LIN {X -0.031,Y -424.133,Z 625.479,A 0.000,B 0.000,C 90.000,E1 266.216} C_DIS
LIN {X -0.178,Y -415.760,Z 625.479,A 0.000,B 0.000,C 90.000,E1 266.159} C_DIS
LIN {X 0.095,Y -410.358,Z 625.478,A 0.000,B 0.000,C 90.000,E1 266.102} C_DIS
LIN {X 0.011,Y -180.925,Z 625.478,A 0.000,B 0.000,C 90.000,E1 266.102} C_DIS
LIN {X -0.004,Y -180.875,Z 625.473,A 0.000,B 0.000,C 90.000,E1 265.065} C_DIS
LIN {X 0.078,Y -178.941,Z 625.443,A 0.000,B 0.000,C 90.000,E1 259.803} C_DIS
LIN {X -0.054,Y -175.991,Z 625.415,A 0.000,B 0.000,C 90.000,E1 254.755} C_DIS
LIN {X 0.061,Y -175.493,Z 625.410,A 0.000,B 0.000,C 90.000,E1 253.866} C_DIS
LIN {X -0.045,Y -172.236,Z 625.387,A 0.000,B 0.000,C 90.000,E1 249.625} C_DIS
LIN {X -0.066,Y -171.714,Z 625.382,A 0.000,B 0.000,C 90.000,E1 248.773} C_DIS
LIN {X 0.019,Y -167.309,Z 625.353,A 0.000,B 0.000,C 90.000,E1 243.563} C_DIS
LIN {X 0.024,Y -166.690,Z 625.348,A 0.000,B 0.000,C 90.000,E1 242.692} C_DIS
LIN {X 0.015,Y -162.671,Z 625.324,A 0.000,B 0.000,C 90.000,E1 238.329} C_DIS
LIN {X -0.012,Y -161.361,Z 625.314,A 0.000,B 0.000,C 90.000,E1 236.580} C_DIS
LIN {X 0.022,Y -157.354,Z 625.290,A 0.000,B 0.000,C 90.000,E1 232.145} C_DIS
LIN {X 0.051,Y -155.342,Z 625.275,A 0.000,B 0.000,C 90.000,E1 229.461} C_DIS
LIN {X -0.020,Y -151.690,Z 625.250,A 0.000,B 0.000,C 90.000,E1 225.000} C_DIS
LIN {X 0.028,Y -150.553,Z 625.240,A 0.000,B 0.000,C 90.000,E1 223.176} C_DIS
LIN {X -0.054,Y -147.279,Z 625.215,A 0.000,B 0.000,C 90.000,E1 218.669} C_DIS
LIN {X 0.033,Y -145.307,Z 625.194,A 0.000,B 0.000,C 90.000,E1 214.978} C_DIS
LIN {X 0.025,Y -142.398,Z 625.164,A 0.000,B 0.000,C 90.000,E1 209.461} C_DIS
LIN {X 0.008,Y -141.380,Z 625.148,A 0.000,B 0.000,C 90.000,E1 206.693} C_DIS
LIN {X 0.049,Y -139.349,Z 625.112,A 0.000,B 0.000,C 90.000,E1 200.174} C_DIS
LIN {X -0.009,Y -138.785,Z 625.097,A 0.000,B 0.000,C 90.000,E1 197.402} C_DIS
LIN {X 0.049,Y -138.344,Z 625.055,A 0.000,B 0.000,C 90.000,E1 189.905} C_DIS
LIN {X 0.069,Y -139.387,Z 625.008,A 0.000,B 0.000,C 90.000,E1 181.489} C_DIS
LIN {X -0.017,Y -141.284,Z 624.972,A 0.000,B 0.000,C 90.000,E1 175.008} C_DIS
LIN {X -0.059,Y -142.647,Z 624.957,A 0.000,B 0.000,C 90.000,E1 172.243} C_DIS
LIN {X 0.033,Y -144.984,Z 624.931,A 0.000,B 0.000,C 90.000,E1 167.589} C_DIS
LIN {X 0.023,Y -147.611,Z 624.911,A 0.000,B 0.000,C 90.000,E1 163.921} C_DIS
LIN {X -0.040,Y -150.234,Z 624.890,A 0.000,B 0.000,C 90.000,E1 160.296} C_DIS
LIN {X -0.025,Y -153.627,Z 624.870,A 0.000,B 0.000,C 90.000,E1 156.666} C_DIS
LIN {X -0.037,Y -157.042,Z 624.850,A 0.000,B 0.000,C 90.000,E1 153.076} C_DIS
LIN {X 0.033,Y -161.168,Z 624.831,A 0.000,B 0.000,C 90.000,E1 149.488} C_DIS
LIN {X -0.024,Y -163.264,Z 624.821,A 0.000,B 0.000,C 90.000,E1 147.740} C_DIS
LIN {X 0.074,Y -167.704,Z 624.801,A 0.000,B 0.000,C 90.000,E1 144.196} C_DIS
LIN {X -0.012,Y -171.524,Z 624.787,A 0.000,B 0.000,C 90.000,E1 141.618} C_DIS
LIN {X 0.030,Y -176.462,Z 624.768,A 0.000,B 0.000,C 90.000,E1 138.162} C_DIS
LIN {X -0.099,Y -180.758,Z 624.753,A 0.000,B 0.000,C 90.000,E1 135.648} C_DIS
LIN {X 0.019,Y -186.164,Z 624.735,A 0.000,B 0.000,C 90.000,E1 132.243} C_DIS
LIN {X -0.012,Y -191.121,Z 624.720,A 0.000,B 0.000,C 90.000,E1 129.564} C_DIS
LIN {X -0.069,Y -287.980,Z 624.720,A 0.000,B 0.000,C 90.000,E1 129.564} C_DIS
LIN {X -0.120,Y -289.136,Z 624.720,A 0.000,B 0.000,C 90.000,E1 129.564} C_DIS
LIN {X -0.085,Y -293.449,Z 624.719,A 0.000,B 0.000,C 90.000,E1 129.402} C_DIS
LIN {X 0.178,Y -295.651,Z 624.718,A 0.000,B 0.000,C 90.000,E1 129.197} C_DIS
LIN {X 0.065,Y -298.660,Z 624.716,A 0.000,B 0.000,C 90.000,E1 128.910} C_DIS
LIN {X 0.032,Y -302.298,Z 624.713,A 0.000,B 0.000,C 90.000,E1 128.338} C_DIS
LIN {X -0.020,Y -303.752,Z 624.711,A 0.000,B 0.000,C 90.000,E1 128.016} C_DIS
LIN {X -0.020,Y -304.897,Z 624.709,A 0.000,B 0.000,C 90.000,E1 127.684} C_DIS
LIN {X 0.096,Y -315.476,Z 624.689,A 0.000,B 0.000,C 90.000,E1 124.072} C_DIS
LIN {X -0.022,Y -325.465,Z 624.673,A 0.000,B 0.000,C 90.000,E1 121.209} C_DIS
LIN {X 0.087,Y -336.777,Z 624.658,A 0.000,B 0.000,C 90.000,E1 118.359} C_DIS
LIN {X 0.035,Y -349.518,Z 624.642,A 0.000,B 0.000,C 90.000,E1 115.591} C_DIS
LIN {X -0.166,Y -362.130,Z 624.629,A 0.000,B 0.000,C 90.000,E1 113.206} C_DIS
LIN {X 0.145,Y -376.051,Z 624.616,A 0.000,B 0.000,C 90.000,E1 110.791} C_DIS
LIN {X 0.066,Y -391.379,Z 624.603,A 0.000,B 0.000,C 90.000,E1 108.489} C_DIS
LIN {X -0.135,Y -408.226,Z 624.590,A 0.000,B 0.000,C 90.000,E1 106.260} C_DIS
LIN {X -0.165,Y -426.717,Z 624.578,A 0.000,B 0.000,C 90.000,E1 104.064} C_DIS
LIN {X -0.079,Y -446.611,Z 624.566,A 0.000,B 0.000,C 90.000,E1 101.951} C_DIS
LIN {X -0.051,Y -467.104,Z 624.556,A 0.000,B 0.000,C 90.000,E1 100.018} C_DIS
LIN {X -0.014,Y -472.187,Z 624.553,A 0.000,B 0.000,C 90.000,E1 99.557} C_DIS
LIN {X 0.000,Y -474.149,Z 624.552,A 0.000,B 0.000,C 90.000,E1 99.321} C_DIS
LIN {X -0.064,Y -475.647,Z 624.550,A 0.000,B 0.000,C 90.000,E1 99.095} C_DIS
LIN {X -0.200,Y -476.871,Z 624.549,A 0.000,B 0.000,C 90.000,E1 98.859} C_DIS
LIN {X 0.135,Y -477.767,Z 624.548,A 0.000,B 0.000,C 90.000,E1 98.568} C_DIS
LIN {X -0.197,Y -478.729,Z 624.545,A 0.000,B 0.000,C 90.000,E1 98.106} C_DIS
LIN {X -0.049,Y -478.707,Z 624.542,A 0.000,B 0.000,C 90.000,E1 97.587} C_DIS
LIN {X 0.106,Y -477.700,Z 624.539,A 0.000,B 0.000,C 90.000,E1 97.068} C_DIS
LIN {X -0.024,Y -476.783,Z 624.538,A 0.000,B 0.000,C 90.000,E1 96.834} C_DIS
LIN {X -0.212,Y -475.534,Z 624.537,A 0.000,B 0.000,C 90.000,E1 96.606} C_DIS
LIN {X -0.214,Y -470.227,Z 624.532,A 0.000,B 0.000,C 90.000,E1 95.853} C_DIS
LIN {X 0.070,Y -456.360,Z 624.521,A 0.000,B 0.000,C 90.000,E1 93.784} C_DIS
LIN {X 0.196,Y -442.672,Z 624.508,A 0.000,B 0.000,C 90.000,E1 91.432} C_DIS
LIN {X 0.081,Y -432.630,Z 624.498,A 0.000,B 0.000,C 90.000,E1 89.599} C_DIS
LIN {X -0.058,Y -425.082,Z 624.490,A 0.000,B 0.000,C 90.000,E1 88.282} C_DIS
LIN {X -0.169,Y -415.676,Z 624.481,A 0.000,B 0.000,C 90.000,E1 86.674} C_DIS
LIN {X -0.133,Y -400.162,Z 624.466,A 0.000,B 0.000,C 90.000,E1 83.913} C_DIS
LIN {X -0.126,Y -386.762,Z 624.452,A 0.000,B 0.000,C 90.000,E1 81.376} C_DIS
LIN {X 0.075,Y -372.503,Z 624.436,A 0.000,B 0.000,C 90.000,E1 78.465} C_DIS
LIN {X 0.060,Y -361.513,Z 624.423,A 0.000,B 0.000,C 90.000,E1 76.117} C_DIS
LIN {X -0.050,Y -347.259,Z 624.405,A 0.000,B 0.000,C 90.000,E1 72.834} C_DIS
LIN {X 0.039,Y -336.337,Z 624.389,A 0.000,B 0.000,C 90.000,E1 70.061} C_DIS
LIN {X 0.095,Y -324.067,Z 624.370,A 0.000,B 0.000,C 90.000,E1 66.613} C_DIS
LIN {X -0.068,Y -314.012,Z 624.352,A 0.000,B 0.000,C 90.000,E1 63.461} C_DIS
LIN {X 0.025,Y -304.661,Z 624.334,A 0.000,B 0.000,C 90.000,E1 60.205} C_DIS
LIN {X 0.025,Y -295.894,Z 624.316,A 0.000,B 0.000,C 90.000,E1 56.914} C_DIS
LIN {X -0.010,Y -287.671,Z 624.298,A 0.000,B 0.000,C 90.000,E1 53.577} C_DIS
LIN {X -0.099,Y -281.225,Z 624.283,A 0.000,B 0.000,C 90.000,E1 50.884} C_DIS
LIN {X 0.000,Y -276.089,Z 624.271,A 0.000,B 0.000,C 90.000,E1 48.809} C_DIS
LIN {X 0.175,Y -272.365,Z 624.263,A 0.000,B 0.000,C 90.000,E1 47.391} C_DIS
LIN {X -0.075,Y -268.402,Z 624.256,A 0.000,B 0.000,C 90.000,E1 46.053} C_DIS
LIN {X -0.067,Y -261.947,Z 624.244,A 0.000,B 0.000,C 90.000,E1 43.947} C_DIS
LIN {X 0.019,Y -253.976,Z 624.230,A 0.000,B 0.000,C 90.000,E1 41.434} C_DIS
LIN {X -0.009,Y -244.166,Z 624.212,A 0.000,B 0.000,C 90.000,E1 38.177} C_DIS
LIN {X -0.027,Y -236.115,Z 624.196,A 0.000,B 0.000,C 90.000,E1 35.231} C_DIS
LIN {X 0.061,Y -228.843,Z 624.179,A 0.000,B 0.000,C 90.000,E1 32.212} C_DIS
LIN {X 0.032,Y -220.667,Z 624.158,A 0.000,B 0.000,C 90.000,E1 28.409} C_DIS
LIN {X -0.044,Y -214.977,Z 624.141,A 0.000,B 0.000,C 90.000,E1 25.335} C_DIS
LIN {X -0.012,Y -208.974,Z 624.119,A 0.000,B 0.000,C 90.000,E1 21.408} C_DIS
LIN {X -0.072,Y -204.153,Z 624.097,A 0.000,B 0.000,C 90.000,E1 17.457} C_DIS
LIN {X 0.061,Y -200.407,Z 624.075,A 0.000,B 0.000,C 90.000,E1 13.411} C_DIS
LIN {X 0.038,Y -197.242,Z 624.048,A 0.000,B 0.000,C 90.000,E1 8.568} C_DIS
LIN {X 0.032,Y -197.987,Z 623.952,A 0.000,B 0.000,C 90.000,E1 351.376} C_DIS
LIN {X 0.025,Y -201.441,Z 623.925,A 0.000,B 0.000,C 90.000,E1 346.520} C_DIS
LIN {X 0.072,Y -205.463,Z 623.903,A 0.000,B 0.000,C 90.000,E1 342.489} C_DIS
LIN {X -0.041,Y -210.309,Z 623.881,A 0.000,B 0.000,C 90.000,E1 338.539} C_DIS
LIN {X 0.002,Y -215.908,Z 623.859,A 0.000,B 0.000,C 90.000,E1 334.588} C_DIS
LIN {X -0.073,Y -222.153,Z 623.837,A 0.000,B 0.000,C 90.000,E1 330.717} C_DIS
LIN {X 0.101,Y -229.051,Z 623.816,A 0.000,B 0.000,C 90.000,E1 326.834} C_DIS
LIN {X -0.003,Y -235.031,Z 623.799,A 0.000,B 0.000,C 90.000,E1 323.829} C_DIS
LIN {X 0.095,Y -242.933,Z 623.778,A 0.000,B 0.000,C 90.000,E1 320.070} C_DIS
LIN {X -0.013,Y -251.590,Z 623.758,A 0.000,B 0.000,C 90.000,E1 316.419} C_DIS
LIN {X -0.035,Y -261.286,Z 623.738,A 0.000,B 0.000,C 90.000,E1 312.813} C_DIS
LIN {X 0.019,Y -270.004,Z 623.722,A 0.000,B 0.000,C 90.000,E1 309.967} C_DIS
LIN {X -0.030,Y -282.468,Z 623.703,A 0.000,B 0.000,C 90.000,E1 306.503} C_DIS
LIN {X 0.103,Y -296.445,Z 623.684,A 0.000,B 0.000,C 90.000,E1 303.086} C_DIS
LIN {X 0.049,Y -312.049,Z 623.666,A 0.000,B 0.000,C 90.000,E1 299.795} C_DIS
LIN {X -0.073,Y -327.245,Z 623.649,A 0.000,B 0.000,C 90.000,E1 296.924} C_DIS
LIN {X 0.087,Y -344.942,Z 623.632,A 0.000,B 0.000,C 90.000,E1 293.770} C_DIS
LIN {X -0.016,Y -360.212,Z 623.619,A 0.000,B 0.000,C 90.000,E1 291.354} C_DIS
LIN {X 0.111,Y -378.973,Z 623.604,A 0.000,B 0.000,C 90.000,E1 288.671} C_DIS
LIN {X 0.178,Y -399.589,Z 623.589,A 0.000,B 0.000,C 90.000,E1 286.079} C_DIS
LIN {X 0.017,Y -413.489,Z 623.580,A 0.000,B 0.000,C 90.000,E1 284.426} C_DIS
LIN {X -0.050,Y -424.647,Z 623.573,A 0.000,B 0.000,C 90.000,E1 283.063} C_DIS
LIN {X -0.045,Y -435.361,Z 623.565,A 0.000,B 0.000,C 90.000,E1 281.715} C_DIS
LIN {X 0.112,Y -445.670,Z 623.558,A 0.000,B 0.000,C 90.000,E1 280.366} C_DIS
LIN {X 0.083,Y -457.496,Z 623.549,A 0.000,B 0.000,C 90.000,E1 278.803} C_DIS
LIN {X -0.025,Y -466.986,Z 623.542,A 0.000,B 0.000,C 90.000,E1 277.530} C_DIS
LIN {X -0.112,Y -472.142,Z 623.538,A 0.000,B 0.000,C 90.000,E1 276.777} C_DIS
LIN {X -0.006,Y -475.183,Z 623.535,A 0.000,B 0.000,C 90.000,E1 276.258} C_DIS
LIN {X 0.120,Y -477.839,Z 623.532,A 0.000,B 0.000,C 90.000,E1 275.739} C_DIS
LIN {X -0.215,Y -480.121,Z 623.529,A 0.000,B 0.000,C 90.000,E1 275.277} C_DIS
LIN {X -0.062,Y -482.024,Z 623.526,A 0.000,B 0.000,C 90.000,E1 274.759} C_DIS
LIN {X 0.062,Y -483.545,Z 623.524,A 0.000,B 0.000,C 90.000,E1 274.245} C_DIS
LIN {X 0.234,Y -484.683,Z 623.521,A 0.000,B 0.000,C 90.000,E1 273.726} C_DIS
LIN {X -0.100,Y -485.485,Z 623.518,A 0.000,B 0.000,C 90.000,E1 273.269} C_DIS
LIN {X 0.084,Y -485.991,Z 623.515,A 0.000,B 0.000,C 90.000,E1 272.751} C_DIS
LIN {X -0.237,Y -486.190,Z 623.513,A 0.000,B 0.000,C 90.000,E1 272.293} C_DIS
LIN {X -0.051,Y -486.080,Z 623.510,A 0.000,B 0.000,C 90.000,E1 271.776} C_DIS
LIN {X 0.118,Y -485.598,Z 623.507,A 0.000,B 0.000,C 90.000,E1 271.260} C_DIS
LIN {X -0.196,Y -484.736,Z 623.504,A 0.000,B 0.000,C 90.000,E1 270.802} C_DIS
LIN {X -0.027,Y -483.413,Z 623.502,A 0.000,B 0.000,C 90.000,E1 270.286} C_DIS
LIN {X 0.136,Y -481.532,Z 623.499,A 0.000,B 0.000,C 90.000,E1 269.771} C_DIS
LIN {X -0.189,Y -478.902,Z 623.496,A 0.000,B 0.000,C 90.000,E1 269.312} C_DIS
LIN {X 0.118,Y -477.369,Z 623.495,A 0.000,B 0.000,C 90.000,E1 269.026} C_DIS
LIN {X -0.230,Y -473.473,Z 623.492,A 0.000,B 0.000,C 90.000,E1 268.568} C_DIS
LIN {X 0.064,Y -471.160,Z 623.490,A 0.000,B 0.000,C 90.000,E1 268.282} C_DIS
LIN {X -0.109,Y -468.523,Z 623.489,A 0.000,B 0.000,C 90.000,E1 268.051} C_DIS
LIN {X 0.217,Y -462.608,Z 623.486,A 0.000,B 0.000,C 90.000,E1 267.535} C_DIS
LIN {X -0.198,Y -459.195,Z 623.485,A 0.000,B 0.000,C 90.000,E1 267.364} C_DIS
LIN {X 0.042,Y -452.155,Z 623.483,A 0.000,B 0.000,C 90.000,E1 266.963} C_DIS
LIN {X 0.003,Y -444.697,Z 623.482,A 0.000,B 0.000,C 90.000,E1 266.674} C_DIS
LIN {X 0.010,Y -437.024,Z 623.480,A 0.000,B 0.000,C 90.000,E1 266.445} C_DIS
LIN {X 0.005,Y -428.475,Z 623.479,A 0.000,B 0.000,C 90.000,E1 266.274} C_DIS
LIN {X -0.014,Y -419.041,Z 623.479,A 0.000,B 0.000,C 90.000,E1 266.159} C_DIS
LIN {X 0.112,Y -411.810,Z 623.478,A 0.000,B 0.000,C 90.000,E1 266.102} C_DIS
LIN {X 0.018,Y -180.925,Z 623.478,A 0.000,B 0.000,C 90.000,E1 266.102} C_DIS
LIN {X -0.019,Y -180.899,Z 623.474,A 0.000,B 0.000,C 90.000,E1 265.241} C_DIS
LIN {X -0.069,Y -180.215,Z 623.464,A 0.000,B 0.000,C 90.000,E1 263.571} C_DIS
LIN {X 0.061,Y -179.034,Z 623.445,A 0.000,B 0.000,C 90.000,E1 260.151} C_DIS
LIN {X -0.052,Y -178.692,Z 623.441,A 0.000,B 0.000,C 90.000,E1 259.342} C_DIS
LIN {X 0.057,Y -175.741,Z 623.412,A 0.000,B 0.000,C 90.000,E1 254.212} C_DIS
LIN {X 0.053,Y -171.925,Z 623.384,A 0.000,B 0.000,C 90.000,E1 249.082} C_DIS
LIN {X 0.028,Y -171.298,Z 623.379,A 0.000,B 0.000,C 90.000,E1 248.230} C_DIS
LIN {X 0.073,Y -167.560,Z 623.355,A 0.000,B 0.000,C 90.000,E1 243.896} C_DIS
LIN {X 0.086,Y -166.186,Z 623.345,A 0.000,B 0.000,C 90.000,E1 242.153} C_DIS
LIN {X 0.076,Y -162.955,Z 623.326,A 0.000,B 0.000,C 90.000,E1 238.663} C_DIS
LIN {X -0.100,Y -160.863,Z 623.311,A 0.000,B 0.000,C 90.000,E1 236.087} C_DIS
LIN {X 0.100,Y -157.638,Z 623.292,A 0.000,B 0.000,C 90.000,E1 232.477} C_DIS
LIN {X 0.038,Y -155.676,Z 623.277,A 0.000,B 0.000,C 90.000,E1 229.828} C_DIS
LIN {X -0.017,Y -151.943,Z 623.252,A 0.000,B 0.000,C 90.000,E1 225.364} C_DIS
LIN {X -0.006,Y -150.181,Z 623.237,A 0.000,B 0.000,C 90.000,E1 222.651} C_DIS
LIN {X 0.023,Y -146.955,Z 623.212,A 0.000,B 0.000,C 90.000,E1 218.096} C_DIS
LIN {X 0.011,Y -145.542,Z 623.196,A 0.000,B 0.000,C 90.000,E1 215.358} C_DIS
LIN {X -0.072,Y -142.938,Z 623.171,A 0.000,B 0.000,C 90.000,E1 210.797} C_DIS
LIN {X -0.015,Y -141.562,Z 623.150,A 0.000,B 0.000,C 90.000,E1 207.078} C_DIS
LIN {X 0.037,Y -139.409,Z 623.114,A 0.000,B 0.000,C 90.000,E1 200.556} C_DIS
LIN {X -0.041,Y -139.131,Z 623.104,A 0.000,B 0.000,C 90.000,E1 198.725} C_DIS
LIN {X -0.014,Y -138.350,Z 623.057,A 0.000,B 0.000,C 90.000,E1 190.310} C_DIS
LIN {X -0.026,Y -139.498,Z 623.005,A 0.000,B 0.000,C 90.000,E1 180.974} C_DIS
LIN {X 0.054,Y -141.118,Z 622.974,A 0.000,B 0.000,C 90.000,E1 175.355} C_DIS
LIN {X 0.008,Y -142.499,Z 622.959,A 0.000,B 0.000,C 90.000,E1 172.591} C_DIS
LIN {X -0.046,Y -144.753,Z 622.933,A 0.000,B 0.000,C 90.000,E1 167.993} C_DIS
LIN {X 0.047,Y -147.362,Z 622.913,A 0.000,B 0.000,C 90.000,E1 164.283} C_DIS
LIN {X -0.032,Y -150.689,Z 622.887,A 0.000,B 0.000,C 90.000,E1 159.752} C_DIS
LIN {X 0.051,Y -154.169,Z 622.867,A 0.000,B 0.000,C 90.000,E1 156.102} C_DIS
LIN {X -0.018,Y -157.603,Z 622.847,A 0.000,B 0.000,C 90.000,E1 152.538} C_DIS
LIN {X -0.068,Y -161.855,Z 622.828,A 0.000,B 0.000,C 90.000,E1 148.997} C_DIS
LIN {X -0.050,Y -166.045,Z 622.808,A 0.000,B 0.000,C 90.000,E1 145.468} C_DIS
LIN {X -0.060,Y -171.049,Z 622.789,A 0.000,B 0.000,C 90.000,E1 141.984} C_DIS
LIN {X -0.029,Y -175.920,Z 622.770,A 0.000,B 0.000,C 90.000,E1 138.528} C_DIS
LIN {X -0.037,Y -180.159,Z 622.755,A 0.000,B 0.000,C 90.000,E1 135.972} C_DIS
LIN {X -0.068,Y -185.576,Z 622.737,A 0.000,B 0.000,C 90.000,E1 132.609} C_DIS
LIN {X -0.047,Y -191.138,Z 622.720,A 0.000,B 0.000,C 90.000,E1 129.564} C_DIS
LIN {X -0.124,Y -288.693,Z 622.720,A 0.000,B 0.000,C 90.000,E1 129.564} C_DIS
LIN {X 0.047,Y -289.451,Z 622.720,A 0.000,B 0.000,C 90.000,E1 129.519} C_DIS
LIN {X -0.100,Y -295.241,Z 622.718,A 0.000,B 0.000,C 90.000,E1 129.277} C_DIS
LIN {X 0.061,Y -298.242,Z 622.716,A 0.000,B 0.000,C 90.000,E1 128.955} C_DIS
LIN {X 0.157,Y -301.914,Z 622.713,A 0.000,B 0.000,C 90.000,E1 128.382} C_DIS
LIN {X -0.084,Y -303.451,Z 622.712,A 0.000,B 0.000,C 90.000,E1 128.096} C_DIS
LIN {X 0.102,Y -304.661,Z 622.710,A 0.000,B 0.000,C 90.000,E1 127.729} C_DIS
LIN {X -0.003,Y -316.286,Z 622.688,A 0.000,B 0.000,C 90.000,E1 123.833} C_DIS
LIN {X 0.167,Y -326.386,Z 622.672,A 0.000,B 0.000,C 90.000,E1 120.924} C_DIS
LIN {X 0.137,Y -337.822,Z 622.656,A 0.000,B 0.000,C 90.000,E1 118.103} C_DIS
LIN {X 0.122,Y -350.690,Z 622.641,A 0.000,B 0.000,C 90.000,E1 115.335} C_DIS
LIN {X -0.049,Y -363.428,Z 622.627,A 0.000,B 0.000,C 90.000,E1 112.950} C_DIS
LIN {X -0.190,Y -377.482,Z 622.614,A 0.000,B 0.000,C 90.000,E1 110.610} C_DIS
LIN {X -0.121,Y -392.955,Z 622.602,A 0.000,B 0.000,C 90.000,E1 108.290} C_DIS
LIN {X -0.027,Y -409.960,Z 622.589,A 0.000,B 0.000,C 90.000,E1 106.024} C_DIS
LIN {X -0.008,Y -428.620,Z 622.577,A 0.000,B 0.000,C 90.000,E1 103.828} C_DIS
LIN {X -0.222,Y -448.583,Z 622.565,A 0.000,B 0.000,C 90.000,E1 101.771} C_DIS
LIN {X -0.101,Y -471.712,Z 622.553,A 0.000,B 0.000,C 90.000,E1 99.613} C_DIS
LIN {X -0.050,Y -473.785,Z 622.552,A 0.000,B 0.000,C 90.000,E1 99.378} C_DIS
LIN {X -0.077,Y -475.365,Z 622.551,A 0.000,B 0.000,C 90.000,E1 99.151} C_DIS
LIN {X -0.214,Y -476.688,Z 622.549,A 0.000,B 0.000,C 90.000,E1 98.916} C_DIS
LIN {X 0.119,Y -477.667,Z 622.548,A 0.000,B 0.000,C 90.000,E1 98.624} C_DIS
LIN {X -0.215,Y -478.768,Z 622.545,A 0.000,B 0.000,C 90.000,E1 98.163} C_DIS
LIN {X -0.068,Y -478.874,Z 622.542,A 0.000,B 0.000,C 90.000,E1 97.644} C_DIS
LIN {X 0.087,Y -478.002,Z 622.540,A 0.000,B 0.000,C 90.000,E1 97.125} C_DIS
LIN {X -0.231,Y -476.007,Z 622.537,A 0.000,B 0.000,C 90.000,E1 96.663} C_DIS
LIN {X 0.108,Y -474.463,Z 622.535,A 0.000,B 0.000,C 90.000,E1 96.372} C_DIS
LIN {X -0.195,Y -458.525,Z 622.523,A 0.000,B 0.000,C 90.000,E1 94.131} C_DIS
LIN {X -0.194,Y -446.005,Z 622.511,A 0.000,B 0.000,C 90.000,E1 92.064} C_DIS
LIN {X -0.055,Y -434.514,Z 622.500,A 0.000,B 0.000,C 90.000,E1 89.943} C_DIS
LIN {X -0.168,Y -427.077,Z 622.492,A 0.000,B 0.000,C 90.000,E1 88.625} C_DIS
LIN {X 0.153,Y -417.704,Z 622.483,A 0.000,B 0.000,C 90.000,E1 86.963} C_DIS
LIN {X 0.175,Y -403.651,Z 622.470,A 0.000,B 0.000,C 90.000,E1 84.489} C_DIS
LIN {X -0.115,Y -388.651,Z 622.454,A 0.000,B 0.000,C 90.000,E1 81.724} C_DIS
LIN {X 0.142,Y -374.339,Z 622.438,A 0.000,B 0.000,C 90.000,E1 78.814} C_DIS
LIN {X 0.142,Y -361.902,Z 622.423,A 0.000,B 0.000,C 90.000,E1 76.172} C_DIS
LIN {X -0.055,Y -347.621,Z 622.405,A 0.000,B 0.000,C 90.000,E1 72.906} C_DIS
LIN {X 0.035,Y -336.702,Z 622.390,A 0.000,B 0.000,C 90.000,E1 70.134} C_DIS
LIN {X -0.077,Y -324.414,Z 622.371,A 0.000,B 0.000,C 90.000,E1 66.719} C_DIS
LIN {X 0.070,Y -314.374,Z 622.353,A 0.000,B 0.000,C 90.000,E1 63.512} C_DIS
LIN {X 0.028,Y -305.013,Z 622.335,A 0.000,B 0.000,C 90.000,E1 60.284} C_DIS
LIN {X 0.033,Y -296.225,Z 622.317,A 0.000,B 0.000,C 90.000,E1 56.993} C_DIS
LIN {X 0.174,Y -287.979,Z 622.298,A 0.000,B 0.000,C 90.000,E1 53.623} C_DIS
LIN {X 0.053,Y -283.148,Z 622.287,A 0.000,B 0.000,C 90.000,E1 51.618} C_DIS
LIN {X -0.022,Y -278.181,Z 622.275,A 0.000,B 0.000,C 90.000,E1 49.585} C_DIS
LIN {X 0.000,Y -272.685,Z 622.264,A 0.000,B 0.000,C 90.000,E1 47.514} C_DIS
LIN {X -0.047,Y -268.728,Z 622.256,A 0.000,B 0.000,C 90.000,E1 46.134} C_DIS
LIN {X -0.150,Y -264.525,Z 622.248,A 0.000,B 0.000,C 90.000,E1 44.757} C_DIS
LIN {X -0.032,Y -257.787,Z 622.237,A 0.000,B 0.000,C 90.000,E1 42.609} C_DIS
LIN {X -0.006,Y -248.806,Z 622.221,A 0.000,B 0.000,C 90.000,E1 39.725} C_DIS
LIN {X 0.040,Y -240.382,Z 622.204,A 0.000,B 0.000,C 90.000,E1 36.790} C_DIS
LIN {X -0.023,Y -232.669,Z 622.188,A 0.000,B 0.000,C 90.000,E1 33.833} C_DIS
LIN {X 0.047,Y -225.733,Z 622.171,A 0.000,B 0.000,C 90.000,E1 30.797} C_DIS
LIN {X -0.086,Y -219.430,Z 622.154,A 0.000,B 0.000,C 90.000,E1 27.769} C_DIS
LIN {X 0.006,Y -213.907,Z 622.137,A 0.000,B 0.000,C 90.000,E1 24.643} C_DIS
LIN {X -0.073,Y -208.089,Z 622.115,A 0.000,B 0.000,C 90.000,E1 20.737} C_DIS
LIN {X 0.035,Y -203.445,Z 622.093,A 0.000,B 0.000,C 90.000,E1 16.732} C_DIS
LIN {X 0.044,Y -199.910,Z 622.071,A 0.000,B 0.000,C 90.000,E1 12.715} C_DIS
LIN {X 0.008,Y -196.965,Z 622.044,A 0.000,B 0.000,C 90.000,E1 7.871} C_DIS
LIN {X 0.035,Y -198.041,Z 621.952,A 0.000,B 0.000,C 90.000,E1 351.376} C_DIS
LIN {X 0.030,Y -201.501,Z 621.925,A 0.000,B 0.000,C 90.000,E1 346.520} C_DIS
LIN {X 0.079,Y -205.521,Z 621.903,A 0.000,B 0.000,C 90.000,E1 342.489} C_DIS
LIN {X -0.032,Y -210.373,Z 621.881,A 0.000,B 0.000,C 90.000,E1 338.539} C_DIS
LIN {X 0.014,Y -215.948,Z 621.859,A 0.000,B 0.000,C 90.000,E1 334.588} C_DIS
LIN {X -0.059,Y -222.182,Z 621.837,A 0.000,B 0.000,C 90.000,E1 330.717} C_DIS
LIN {X 0.115,Y -229.089,Z 621.816,A 0.000,B 0.000,C 90.000,E1 326.834} C_DIS
LIN {X 0.013,Y -235.054,Z 621.799,A 0.000,B 0.000,C 90.000,E1 323.829} C_DIS
LIN {X 0.112,Y -242.941,Z 621.778,A 0.000,B 0.000,C 90.000,E1 320.070} C_DIS
LIN {X 0.004,Y -251.552,Z 621.758,A 0.000,B 0.000,C 90.000,E1 316.419} C_DIS
LIN {X -0.025,Y -261.222,Z 621.738,A 0.000,B 0.000,C 90.000,E1 312.813} C_DIS
LIN {X 0.028,Y -269.921,Z 621.722,A 0.000,B 0.000,C 90.000,E1 309.967} C_DIS
LIN {X -0.023,Y -282.393,Z 621.703,A 0.000,B 0.000,C 90.000,E1 306.503} C_DIS
LIN {X 0.106,Y -296.363,Z 621.684,A 0.000,B 0.000,C 90.000,E1 303.086} C_DIS
LIN {X 0.050,Y -311.953,Z 621.666,A 0.000,B 0.000,C 90.000,E1 299.795} C_DIS
LIN {X -0.164,Y -325.407,Z 621.651,A 0.000,B 0.000,C 90.000,E1 297.257} C_DIS
LIN {X 0.080,Y -343.002,Z 621.634,A 0.000,B 0.000,C 90.000,E1 294.079} C_DIS
LIN {X -0.023,Y -360.116,Z 621.619,A 0.000,B 0.000,C 90.000,E1 291.354} C_DIS
LIN {X 0.102,Y -378.930,Z 621.604,A 0.000,B 0.000,C 90.000,E1 288.671} C_DIS
LIN {X 0.166,Y -399.578,Z 621.589,A 0.000,B 0.000,C 90.000,E1 286.079} C_DIS
LIN {X 0.004,Y -413.468,Z 621.580,A 0.000,B 0.000,C 90.000,E1 284.426} C_DIS
LIN {X 0.094,Y -426.825,Z 621.571,A 0.000,B 0.000,C 90.000,E1 282.771} C_DIS
LIN {X 0.130,Y -437.439,Z 621.564,A 0.000,B 0.000,C 90.000,E1 281.422} C_DIS
LIN {X 0.098,Y -445.695,Z 621.558,A 0.000,B 0.000,C 90.000,E1 280.366} C_DIS
LIN {X -0.187,Y -455.511,Z 621.550,A 0.000,B 0.000,C 90.000,E1 279.095} C_DIS
LIN {X 0.191,Y -465.060,Z 621.543,A 0.000,B 0.000,C 90.000,E1 277.757} C_DIS
LIN {X 0.093,Y -470.431,Z 621.539,A 0.000,B 0.000,C 90.000,E1 277.004} C_DIS
LIN {X -0.023,Y -475.070,Z 621.535,A 0.000,B 0.000,C 90.000,E1 276.258} C_DIS
LIN {X 0.102,Y -477.718,Z 621.532,A 0.000,B 0.000,C 90.000,E1 275.739} C_DIS
LIN {X 0.243,Y -480.022,Z 621.529,A 0.000,B 0.000,C 90.000,E1 275.220} C_DIS
LIN {X -0.081,Y -481.915,Z 621.526,A 0.000,B 0.000,C 90.000,E1 274.759} C_DIS
LIN {X 0.042,Y -483.462,Z 621.524,A 0.000,B 0.000,C 90.000,E1 274.245} C_DIS
LIN {X 0.214,Y -484.633,Z 621.521,A 0.000,B 0.000,C 90.000,E1 273.726} C_DIS
LIN {X -0.121,Y -485.457,Z 621.518,A 0.000,B 0.000,C 90.000,E1 273.269} C_DIS
LIN {X 0.063,Y -485.979,Z 621.515,A 0.000,B 0.000,C 90.000,E1 272.751} C_DIS
LIN {X 0.227,Y -486.160,Z 621.513,A 0.000,B 0.000,C 90.000,E1 272.236} C_DIS
LIN {X -0.072,Y -486.039,Z 621.510,A 0.000,B 0.000,C 90.000,E1 271.776} C_DIS
LIN {X 0.097,Y -485.626,Z 621.507,A 0.000,B 0.000,C 90.000,E1 271.260} C_DIS
LIN {X -0.217,Y -484.749,Z 621.504,A 0.000,B 0.000,C 90.000,E1 270.802} C_DIS
LIN {X -0.048,Y -483.438,Z 621.502,A 0.000,B 0.000,C 90.000,E1 270.286} C_DIS
LIN {X 0.115,Y -481.512,Z 621.499,A 0.000,B 0.000,C 90.000,E1 269.771} C_DIS
LIN {X -0.210,Y -478.944,Z 621.496,A 0.000,B 0.000,C 90.000,E1 269.312} C_DIS
LIN {X -0.073,Y -475.534,Z 621.493,A 0.000,B 0.000,C 90.000,E1 268.797} C_DIS
LIN {X 0.222,Y -473.538,Z 621.492,A 0.000,B 0.000,C 90.000,E1 268.511} C_DIS
LIN {X -0.129,Y -468.548,Z 621.489,A 0.000,B 0.000,C 90.000,E1 268.051} C_DIS
LIN {X 0.196,Y -462.636,Z 621.486,A 0.000,B 0.000,C 90.000,E1 267.535} C_DIS
LIN {X -0.218,Y -459.197,Z 621.485,A 0.000,B 0.000,C 90.000,E1 267.364} C_DIS
LIN {X 0.139,Y -455.963,Z 621.484,A 0.000,B 0.000,C 90.000,E1 267.135} C_DIS
LIN {X -0.176,Y -448.695,Z 621.482,A 0.000,B 0.000,C 90.000,E1 266.846} C_DIS
LIN {X 0.025,Y -441.247,Z 621.481,A 0.000,B 0.000,C 90.000,E1 266.560} C_DIS
LIN {X -0.201,Y -433.262,Z 621.480,A 0.000,B 0.000,C 90.000,E1 266.388} C_DIS
LIN {X -0.002,Y -424.638,Z 621.479,A 0.000,B 0.000,C 90.000,E1 266.216} C_DIS
LIN {X -0.166,Y -416.410,Z 621.479,A 0.000,B 0.000,C 90.000,E1 266.159} C_DIS
LIN {X 0.102,Y -412.335,Z 621.478,A 0.000,B 0.000,C 90.000,E1 266.102} C_DIS
LIN {X 0.013,Y -180.925,Z 621.478,A 0.000,B 0.000,C 90.000,E1 266.102} C_DIS
LIN {X -0.025,Y -180.899,Z 621.474,A 0.000,B 0.000,C 90.000,E1 265.241} C_DIS
LIN {X -0.075,Y -180.214,Z 621.464,A 0.000,B 0.000,C 90.000,E1 263.571} C_DIS
LIN {X 0.055,Y -179.033,Z 621.445,A 0.000,B 0.000,C 90.000,E1 260.151} C_DIS
LIN {X -0.059,Y -178.690,Z 621.441,A 0.000,B 0.000,C 90.000,E1 259.342} C_DIS
LIN {X 0.052,Y -175.740,Z 621.412,A 0.000,B 0.000,C 90.000,E1 254.212} C_DIS
LIN {X 0.047,Y -171.924,Z 621.384,A 0.000,B 0.000,C 90.000,E1 249.082} C_DIS
LIN {X 0.022,Y -171.296,Z 621.379,A 0.000,B 0.000,C 90.000,E1 248.230} C_DIS
LIN {X 0.067,Y -167.559,Z 621.355,A 0.000,B 0.000,C 90.000,E1 243.896} C_DIS
LIN {X 0.081,Y -166.184,Z 621.345,A 0.000,B 0.000,C 90.000,E1 242.153} C_DIS
LIN {X 0.070,Y -162.954,Z 621.326,A 0.000,B 0.000,C 90.000,E1 238.663} C_DIS
LIN {X -0.106,Y -160.861,Z 621.311,A 0.000,B 0.000,C 90.000,E1 236.087} C_DIS
LIN {X 0.094,Y -157.637,Z 621.292,A 0.000,B 0.000,C 90.000,E1 232.477} C_DIS
LIN {X 0.032,Y -155.674,Z 621.277,A 0.000,B 0.000,C 90.000,E1 229.828} C_DIS
LIN {X 0.084,Y -151.941,Z 621.252,A 0.000,B 0.000,C 90.000,E1 225.324} C_DIS
LIN {X 0.098,Y -150.179,Z 621.237,A 0.000,B 0.000,C 90.000,E1 222.609} C_DIS
LIN {X 0.018,Y -146.954,Z 621.212,A 0.000,B 0.000,C 90.000,E1 218.096} C_DIS
LIN {X 0.006,Y -145.541,Z 621.196,A 0.000,B 0.000,C 90.000,E1 215.358} C_DIS
LIN {X -0.078,Y -142.937,Z 621.171,A 0.000,B 0.000,C 90.000,E1 210.797} C_DIS
LIN {X -0.021,Y -141.561,Z 621.150,A 0.000,B 0.000,C 90.000,E1 207.078} C_DIS
LIN {X 0.032,Y -139.409,Z 621.114,A 0.000,B 0.000,C 90.000,E1 200.556} C_DIS
LIN {X -0.047,Y -139.130,Z 621.104,A 0.000,B 0.000,C 90.000,E1 198.725} C_DIS
LIN {X -0.019,Y -138.350,Z 621.057,A 0.000,B 0.000,C 90.000,E1 190.310} C_DIS
LIN {X -0.031,Y -139.498,Z 621.005,A 0.000,B 0.000,C 90.000,E1 180.974} C_DIS
LIN {X 0.050,Y -141.119,Z 620.974,A 0.000,B 0.000,C 90.000,E1 175.355} C_DIS
LIN {X 0.003,Y -142.499,Z 620.959,A 0.000,B 0.000,C 90.000,E1 172.591} C_DIS
LIN {X -0.050,Y -144.754,Z 620.933,A 0.000,B 0.000,C 90.000,E1 167.993} C_DIS
LIN {X 0.041,Y -147.364,Z 620.913,A 0.000,B 0.000,C 90.000,E1 164.283} C_DIS
LIN {X -0.038,Y -150.691,Z 620.887,A 0.000,B 0.000,C 90.000,E1 159.752} C_DIS
LIN {X 0.045,Y -154.172,Z 620.867,A 0.000,B 0.000,C 90.000,E1 156.102} C_DIS
LIN {X -0.024,Y -157.605,Z 620.847,A 0.000,B 0.000,C 90.000,E1 152.538} C_DIS
LIN {X -0.074,Y -161.857,Z 620.828,A 0.000,B 0.000,C 90.000,E1 148.997} C_DIS
LIN {X -0.057,Y -166.047,Z 620.808,A 0.000,B 0.000,C 90.000,E1 145.468} C_DIS
LIN {X -0.065,Y -171.051,Z 620.789,A 0.000,B 0.000,C 90.000,E1 141.984} C_DIS
LIN {X -0.036,Y -175.924,Z 620.770,A 0.000,B 0.000,C 90.000,E1 138.528} C_DIS
LIN {X -0.044,Y -180.162,Z 620.755,A 0.000,B 0.000,C 90.000,E1 135.972} C_DIS
LIN {X -0.074,Y -185.579,Z 620.737,A 0.000,B 0.000,C 90.000,E1 132.609} C_DIS
LIN {X -0.054,Y -191.142,Z 620.720,A 0.000,B 0.000,C 90.000,E1 129.564} C_DIS
LIN {X -0.134,Y -288.266,Z 620.720,A 0.000,B 0.000,C 90.000,E1 129.564} C_DIS
LIN {X 0.036,Y -289.240,Z 620.720,A 0.000,B 0.000,C 90.000,E1 129.519} C_DIS
LIN {X -0.110,Y -295.190,Z 620.718,A 0.000,B 0.000,C 90.000,E1 129.277} C_DIS
LIN {X -0.097,Y -298.142,Z 620.716,A 0.000,B 0.000,C 90.000,E1 128.991} C_DIS
LIN {X 0.021,Y -301.828,Z 620.713,A 0.000,B 0.000,C 90.000,E1 128.418} C_DIS
LIN {X -0.032,Y -303.383,Z 620.712,A 0.000,B 0.000,C 90.000,E1 128.096} C_DIS
LIN {X 0.153,Y -304.606,Z 620.710,A 0.000,B 0.000,C 90.000,E1 127.729} C_DIS
LIN {X 0.049,Y -316.234,Z 620.688,A 0.000,B 0.000,C 90.000,E1 123.833} C_DIS
LIN {X 0.052,Y -326.330,Z 620.672,A 0.000,B 0.000,C 90.000,E1 120.954} C_DIS
LIN {X -0.108,Y -337.761,Z 620.656,A 0.000,B 0.000,C 90.000,E1 118.153} C_DIS
LIN {X 0.175,Y -350.624,Z 620.641,A 0.000,B 0.000,C 90.000,E1 115.335} C_DIS
LIN {X 0.004,Y -363.357,Z 620.628,A 0.000,B 0.000,C 90.000,E1 112.950} C_DIS
LIN {X -0.137,Y -377.407,Z 620.614,A 0.000,B 0.000,C 90.000,E1 110.610} C_DIS
LIN {X -0.068,Y -392.875,Z 620.602,A 0.000,B 0.000,C 90.000,E1 108.290} C_DIS
LIN {X 0.026,Y -409.873,Z 620.589,A 0.000,B 0.000,C 90.000,E1 106.024} C_DIS
LIN {X 0.045,Y -428.527,Z 620.577,A 0.000,B 0.000,C 90.000,E1 103.828} C_DIS
LIN {X -0.171,Y -448.488,Z 620.565,A 0.000,B 0.000,C 90.000,E1 101.771} C_DIS
LIN {X -0.054,Y -471.632,Z 620.553,A 0.000,B 0.000,C 90.000,E1 99.613} C_DIS
LIN {X 0.004,Y -473.746,Z 620.552,A 0.000,B 0.000,C 90.000,E1 99.378} C_DIS
LIN {X -0.014,Y -475.354,Z 620.551,A 0.000,B 0.000,C 90.000,E1 99.151} C_DIS
LIN {X -0.151,Y -476.707,Z 620.549,A 0.000,B 0.000,C 90.000,E1 98.916} C_DIS
LIN {X 0.181,Y -477.709,Z 620.548,A 0.000,B 0.000,C 90.000,E1 98.624} C_DIS
LIN {X -0.152,Y -478.848,Z 620.545,A 0.000,B 0.000,C 90.000,E1 98.163} C_DIS
LIN {X -0.005,Y -478.990,Z 620.542,A 0.000,B 0.000,C 90.000,E1 97.644} C_DIS
LIN {X 0.150,Y -478.154,Z 620.540,A 0.000,B 0.000,C 90.000,E1 97.125} C_DIS
LIN {X -0.167,Y -476.205,Z 620.537,A 0.000,B 0.000,C 90.000,E1 96.663} C_DIS
LIN {X 0.172,Y -474.692,Z 620.536,A 0.000,B 0.000,C 90.000,E1 96.372} C_DIS
LIN {X -0.128,Y -458.711,Z 620.523,A 0.000,B 0.000,C 90.000,E1 94.131} C_DIS
LIN {X -0.125,Y -446.155,Z 620.511,A 0.000,B 0.000,C 90.000,E1 92.064} C_DIS
LIN {X 0.016,Y -434.662,Z 620.500,A 0.000,B 0.000,C 90.000,E1 89.943} C_DIS
LIN {X -0.096,Y -427.234,Z 620.492,A 0.000,B 0.000,C 90.000,E1 88.625} C_DIS
LIN {X -0.191,Y -417.864,Z 620.483,A 0.000,B 0.000,C 90.000,E1 87.020} C_DIS
LIN {X -0.153,Y -403.799,Z 620.470,A 0.000,B 0.000,C 90.000,E1 84.546} C_DIS
LIN {X -0.039,Y -388.783,Z 620.454,A 0.000,B 0.000,C 90.000,E1 81.724} C_DIS
LIN {X -0.148,Y -374.464,Z 620.438,A 0.000,B 0.000,C 90.000,E1 78.870} C_DIS
LIN {X -0.130,Y -362.035,Z 620.423,A 0.000,B 0.000,C 90.000,E1 76.228} C_DIS
LIN {X 0.024,Y -347.745,Z 620.405,A 0.000,B 0.000,C 90.000,E1 72.906} C_DIS
LIN {X 0.098,Y -334.487,Z 620.386,A 0.000,B 0.000,C 90.000,E1 69.518} C_DIS
LIN {X -0.076,Y -322.495,Z 620.367,A 0.000,B 0.000,C 90.000,E1 66.102} C_DIS
LIN {X 0.142,Y -312.621,Z 620.349,A 0.000,B 0.000,C 90.000,E1 62.871} C_DIS
LIN {X -0.072,Y -303.394,Z 620.331,A 0.000,B 0.000,C 90.000,E1 59.665} C_DIS
LIN {X 0.056,Y -294.657,Z 620.313,A 0.000,B 0.000,C 90.000,E1 56.342} C_DIS
LIN {X -0.013,Y -286.522,Z 620.294,A 0.000,B 0.000,C 90.000,E1 53.004} C_DIS
LIN {X 0.011,Y -281.646,Z 620.283,A 0.000,B 0.000,C 90.000,E1 50.964} C_DIS
LIN {X -0.108,Y -278.310,Z 620.276,A 0.000,B 0.000,C 90.000,E1 49.622} C_DIS
LIN {X -0.091,Y -272.853,Z 620.264,A 0.000,B 0.000,C 90.000,E1 47.553} C_DIS
LIN {X 0.048,Y -268.895,Z 620.256,A 0.000,B 0.000,C 90.000,E1 46.134} C_DIS
LIN {X -0.054,Y -264.668,Z 620.249,A 0.000,B 0.000,C 90.000,E1 44.757} C_DIS
LIN {X 0.063,Y -257.946,Z 620.237,A 0.000,B 0.000,C 90.000,E1 42.609} C_DIS
LIN {X -0.073,Y -246.777,Z 620.217,A 0.000,B 0.000,C 90.000,E1 39.036} C_DIS
LIN {X -0.027,Y -238.503,Z 620.200,A 0.000,B 0.000,C 90.000,E1 36.091} C_DIS
LIN {X 0.058,Y -230.979,Z 620.184,A 0.000,B 0.000,C 90.000,E1 33.086} C_DIS
LIN {X -0.097,Y -222.602,Z 620.163,A 0.000,B 0.000,C 90.000,E1 29.333} C_DIS
LIN {X -0.023,Y -216.663,Z 620.146,A 0.000,B 0.000,C 90.000,E1 26.232} C_DIS
LIN {X -0.047,Y -210.353,Z 620.124,A 0.000,B 0.000,C 90.000,E1 22.333} C_DIS
LIN {X 0.006,Y -205.247,Z 620.102,A 0.000,B 0.000,C 90.000,E1 18.362} C_DIS
LIN {X 0.034,Y -201.238,Z 620.080,A 0.000,B 0.000,C 90.000,E1 14.356} C_DIS
LIN {X 0.082,Y -197.804,Z 620.053,A 0.000,B 0.000,C 90.000,E1 9.500} C_DIS
LIN {X 0.091,Y -195.571,Z 620.012,A 0.000,B 0.000,C 90.000,E1 2.178} C_DIS
LIN {X 0.057,Y -197.284,Z 619.961,A 0.000,B 0.000,C 90.000,E1 352.996} C_DIS
LIN {X -0.098,Y -200.238,Z 619.934,A 0.000,B 0.000,C 90.000,E1 348.173} C_DIS
LIN {X 0.050,Y -203.841,Z 619.912,A 0.000,B 0.000,C 90.000,E1 344.102} C_DIS
LIN {X 0.019,Y -208.390,Z 619.890,A 0.000,B 0.000,C 90.000,E1 340.115} C_DIS
LIN {X -0.047,Y -213.683,Z 619.868,A 0.000,B 0.000,C 90.000,E1 336.177} C_DIS
LIN {X 0.093,Y -219.637,Z 619.846,A 0.000,B 0.000,C 90.000,E1 332.231} C_DIS
LIN {X -0.047,Y -226.298,Z 619.824,A 0.000,B 0.000,C 90.000,E1 328.408} C_DIS
LIN {X -0.076,Y -233.562,Z 619.803,A 0.000,B 0.000,C 90.000,E1 324.609} C_DIS
LIN {X -0.022,Y -241.316,Z 619.782,A 0.000,B 0.000,C 90.000,E1 320.848} C_DIS
LIN {X 0.026,Y -249.729,Z 619.762,A 0.000,B 0.000,C 90.000,E1 317.148} C_DIS
LIN {X -0.060,Y -259.114,Z 619.742,A 0.000,B 0.000,C 90.000,E1 313.542} C_DIS
LIN {X -0.027,Y -268.686,Z 619.724,A 0.000,B 0.000,C 90.000,E1 310.334} C_DIS
LIN {X -0.120,Y -280.992,Z 619.705,A 0.000,B 0.000,C 90.000,E1 306.870} C_DIS
LIN {X -0.036,Y -294.797,Z 619.686,A 0.000,B 0.000,C 90.000,E1 303.452} C_DIS
LIN {X 0.017,Y -310.231,Z 619.667,A 0.000,B 0.000,C 90.000,E1 300.129} C_DIS
LIN {X 0.198,Y -323.590,Z 619.653,A 0.000,B 0.000,C 90.000,E1 297.513} C_DIS
LIN {X 0.092,Y -341.060,Z 619.636,A 0.000,B 0.000,C 90.000,E1 294.387} C_DIS
LIN {X -0.076,Y -358.021,Z 619.620,A 0.000,B 0.000,C 90.000,E1 291.663} C_DIS
LIN {X 0.117,Y -376.678,Z 619.605,A 0.000,B 0.000,C 90.000,E1 288.960} C_DIS
LIN {X 0.161,Y -399.571,Z 619.589,A 0.000,B 0.000,C 90.000,E1 286.079} C_DIS
LIN {X -0.001,Y -413.423,Z 619.580,A 0.000,B 0.000,C 90.000,E1 284.426} C_DIS
LIN {X 0.088,Y -426.821,Z 619.571,A 0.000,B 0.000,C 90.000,E1 282.771} C_DIS
LIN {X 0.123,Y -437.451,Z 619.564,A 0.000,B 0.000,C 90.000,E1 281.422} C_DIS
LIN {X 0.092,Y -445.713,Z 619.558,A 0.000,B 0.000,C 90.000,E1 280.366} C_DIS
LIN {X 0.063,Y -457.427,Z 619.549,A 0.000,B 0.000,C 90.000,E1 278.803} C_DIS
LIN {X 0.183,Y -464.970,Z 619.543,A 0.000,B 0.000,C 90.000,E1 277.757} C_DIS
LIN {X 0.084,Y -470.321,Z 619.539,A 0.000,B 0.000,C 90.000,E1 277.004} C_DIS
LIN {X -0.031,Y -474.954,Z 619.535,A 0.000,B 0.000,C 90.000,E1 276.258} C_DIS
LIN {X -0.098,Y -478.764,Z 619.531,A 0.000,B 0.000,C 90.000,E1 275.511} C_DIS
LIN {X 0.233,Y -479.903,Z 619.529,A 0.000,B 0.000,C 90.000,E1 275.220} C_DIS
LIN {X -0.092,Y -481.845,Z 619.526,A 0.000,B 0.000,C 90.000,E1 274.759} C_DIS
LIN {X 0.030,Y -483.385,Z 619.524,A 0.000,B 0.000,C 90.000,E1 274.245} C_DIS
LIN {X 0.202,Y -484.574,Z 619.521,A 0.000,B 0.000,C 90.000,E1 273.726} C_DIS
LIN {X -0.134,Y -485.426,Z 619.518,A 0.000,B 0.000,C 90.000,E1 273.269} C_DIS
LIN {X 0.050,Y -485.925,Z 619.515,A 0.000,B 0.000,C 90.000,E1 272.751} C_DIS
LIN {X 0.215,Y -486.175,Z 619.513,A 0.000,B 0.000,C 90.000,E1 272.236} C_DIS
LIN {X -0.086,Y -486.033,Z 619.510,A 0.000,B 0.000,C 90.000,E1 271.776} C_DIS
LIN {X 0.084,Y -485.651,Z 619.507,A 0.000,B 0.000,C 90.000,E1 271.260} C_DIS
LIN {X -0.230,Y -484.789,Z 619.504,A 0.000,B 0.000,C 90.000,E1 270.802} C_DIS
LIN {X -0.061,Y -483.430,Z 619.502,A 0.000,B 0.000,C 90.000,E1 270.286} C_DIS
LIN {X 0.102,Y -481.540,Z 619.499,A 0.000,B 0.000,C 90.000,E1 269.771} C_DIS
LIN {X -0.223,Y -478.963,Z 619.496,A 0.000,B 0.000,C 90.000,E1 269.312} C_DIS
LIN {X -0.086,Y -475.553,Z 619.493,A 0.000,B 0.000,C 90.000,E1 268.797} C_DIS
LIN {X 0.031,Y -471.242,Z 619.490,A 0.000,B 0.000,C 90.000,E1 268.282} C_DIS
LIN {X 0.140,Y -465.649,Z 619.488,A 0.000,B 0.000,C 90.000,E1 267.764} C_DIS
LIN {X 0.167,Y -462.605,Z 619.486,A 0.000,B 0.000,C 90.000,E1 267.535} C_DIS
LIN {X 0.192,Y -459.114,Z 619.485,A 0.000,B 0.000,C 90.000,E1 267.306} C_DIS
LIN {X 0.097,Y -455.888,Z 619.484,A 0.000,B 0.000,C 90.000,E1 267.135} C_DIS
LIN {X -0.200,Y -448.660,Z 619.482,A 0.000,B 0.000,C 90.000,E1 266.846} C_DIS
LIN {X 0.016,Y -441.206,Z 619.481,A 0.000,B 0.000,C 90.000,E1 266.560} C_DIS
LIN {X -0.213,Y -433.137,Z 619.480,A 0.000,B 0.000,C 90.000,E1 266.388} C_DIS
LIN {X -0.022,Y -424.341,Z 619.479,A 0.000,B 0.000,C 90.000,E1 266.216} C_DIS
LIN {X 0.082,Y -412.557,Z 619.478,A 0.000,B 0.000,C 90.000,E1 266.102} C_DIS
LIN {X 0.009,Y -407.579,Z 619.478,A 0.000,B 0.000,C 90.000,E1 266.102} C_DIS
LIN {X -0.028,Y -180.924,Z 619.478,A 0.000,B 0.000,C 90.000,E1 266.102} C_DIS
LIN {X -0.035,Y -180.899,Z 619.474,A 0.000,B 0.000,C 90.000,E1 265.241} C_DIS
LIN {X -0.086,Y -180.213,Z 619.464,A 0.000,B 0.000,C 90.000,E1 263.571} C_DIS
LIN {X 0.044,Y -179.033,Z 619.445,A 0.000,B 0.000,C 90.000,E1 260.151} C_DIS
LIN {X -0.069,Y -178.688,Z 619.441,A 0.000,B 0.000,C 90.000,E1 259.342} C_DIS
LIN {X 0.042,Y -175.737,Z 619.412,A 0.000,B 0.000,C 90.000,E1 254.212} C_DIS
LIN {X 0.037,Y -171.921,Z 619.384,A 0.000,B 0.000,C 90.000,E1 249.082} C_DIS
LIN {X 0.012,Y -171.293,Z 619.379,A 0.000,B 0.000,C 90.000,E1 248.230} C_DIS
LIN {X 0.058,Y -167.557,Z 619.355,A 0.000,B 0.000,C 90.000,E1 243.896} C_DIS
LIN {X 0.071,Y -166.180,Z 619.345,A 0.000,B 0.000,C 90.000,E1 242.153} C_DIS
LIN {X 0.060,Y -162.951,Z 619.326,A 0.000,B 0.000,C 90.000,E1 238.663} C_DIS
LIN {X 0.108,Y -160.858,Z 619.311,A 0.000,B 0.000,C 90.000,E1 236.008} C_DIS
LIN {X 0.084,Y -157.634,Z 619.292,A 0.000,B 0.000,C 90.000,E1 232.477} C_DIS
LIN {X 0.023,Y -155.671,Z 619.277,A 0.000,B 0.000,C 90.000,E1 229.828} C_DIS
LIN {X 0.074,Y -151.938,Z 619.252,A 0.000,B 0.000,C 90.000,E1 225.324} C_DIS
LIN {X 0.089,Y -150.176,Z 619.237,A 0.000,B 0.000,C 90.000,E1 222.609} C_DIS
LIN {X 0.009,Y -146.952,Z 619.212,A 0.000,B 0.000,C 90.000,E1 218.096} C_DIS
LIN {X -0.004,Y -145.539,Z 619.196,A 0.000,B 0.000,C 90.000,E1 215.358} C_DIS
LIN {X 0.036,Y -142.935,Z 619.171,A 0.000,B 0.000,C 90.000,E1 210.747} C_DIS
LIN {X -0.030,Y -141.559,Z 619.150,A 0.000,B 0.000,C 90.000,E1 207.078} C_DIS
LIN {X 0.023,Y -139.408,Z 619.114,A 0.000,B 0.000,C 90.000,E1 200.556} C_DIS
LIN {X -0.055,Y -139.129,Z 619.104,A 0.000,B 0.000,C 90.000,E1 198.725} C_DIS
LIN {X -0.028,Y -138.351,Z 619.057,A 0.000,B 0.000,C 90.000,E1 190.310} C_DIS
LIN {X -0.040,Y -139.498,Z 619.005,A 0.000,B 0.000,C 90.000,E1 180.974} C_DIS
LIN {X 0.041,Y -141.121,Z 618.974,A 0.000,B 0.000,C 90.000,E1 175.355} C_DIS
LIN {X -0.006,Y -142.501,Z 618.959,A 0.000,B 0.000,C 90.000,E1 172.591} C_DIS
LIN {X -0.060,Y -144.756,Z 618.933,A 0.000,B 0.000,C 90.000,E1 167.993} C_DIS
LIN {X 0.031,Y -147.367,Z 618.913,A 0.000,B 0.000,C 90.000,E1 164.283} C_DIS
LIN {X -0.046,Y -150.694,Z 618.887,A 0.000,B 0.000,C 90.000,E1 159.752} C_DIS
LIN {X 0.036,Y -154.175,Z 618.867,A 0.000,B 0.000,C 90.000,E1 156.102} C_DIS
LIN {X -0.033,Y -157.609,Z 618.847,A 0.000,B 0.000,C 90.000,E1 152.538} C_DIS
LIN {X 0.055,Y -161.862,Z 618.828,A 0.000,B 0.000,C 90.000,E1 148.948} C_DIS
LIN {X -0.066,Y -166.052,Z 618.808,A 0.000,B 0.000,C 90.000,E1 145.468} C_DIS
LIN {X -0.075,Y -171.056,Z 618.789,A 0.000,B 0.000,C 90.000,E1 141.984} C_DIS
LIN {X -0.046,Y -175.929,Z 618.770,A 0.000,B 0.000,C 90.000,E1 138.528} C_DIS
LIN {X -0.053,Y -180.168,Z 618.755,A 0.000,B 0.000,C 90.000,E1 135.972} C_DIS
LIN {X -0.085,Y -185.585,Z 618.737,A 0.000,B 0.000,C 90.000,E1 132.609} C_DIS
LIN {X -0.101,Y -191.164,Z 618.720,A 0.000,B 0.000,C 90.000,E1 129.564} C_DIS
LIN {X 0.019,Y -289.063,Z 618.720,A 0.000,B 0.000,C 90.000,E1 129.519} C_DIS
LIN {X -0.127,Y -295.151,Z 618.718,A 0.000,B 0.000,C 90.000,E1 129.277} C_DIS
LIN {X -0.081,Y -298.060,Z 618.717,A 0.000,B 0.000,C 90.000,E1 128.991} C_DIS
LIN {X -0.182,Y -301.758,Z 618.714,A 0.000,B 0.000,C 90.000,E1 128.463} C_DIS
LIN {X 0.002,Y -303.327,Z 618.712,A 0.000,B 0.000,C 90.000,E1 128.096} C_DIS
LIN {X 0.188,Y -304.561,Z 618.710,A 0.000,B 0.000,C 90.000,E1 127.729} C_DIS
LIN {X 0.082,Y -316.194,Z 618.688,A 0.000,B 0.000,C 90.000,E1 123.833} C_DIS
LIN {X -0.195,Y -326.287,Z 618.672,A 0.000,B 0.000,C 90.000,E1 121.003} C_DIS
LIN {X -0.075,Y -337.715,Z 618.656,A 0.000,B 0.000,C 90.000,E1 118.153} C_DIS
LIN {X 0.208,Y -350.575,Z 618.641,A 0.000,B 0.000,C 90.000,E1 115.335} C_DIS
LIN {X 0.037,Y -363.305,Z 618.628,A 0.000,B 0.000,C 90.000,E1 112.950} C_DIS
LIN {X -0.104,Y -377.351,Z 618.614,A 0.000,B 0.000,C 90.000,E1 110.610} C_DIS
LIN {X -0.035,Y -392.815,Z 618.602,A 0.000,B 0.000,C 90.000,E1 108.290} C_DIS
LIN {X 0.059,Y -409.810,Z 618.589,A 0.000,B 0.000,C 90.000,E1 106.024} C_DIS
LIN {X 0.078,Y -428.460,Z 618.577,A 0.000,B 0.000,C 90.000,E1 103.828} C_DIS
LIN {X -0.140,Y -448.420,Z 618.565,A 0.000,B 0.000,C 90.000,E1 101.771} C_DIS
LIN {X -0.079,Y -468.963,Z 618.555,A 0.000,B 0.000,C 90.000,E1 99.849} C_DIS
LIN {X -0.025,Y -471.572,Z 618.553,A 0.000,B 0.000,C 90.000,E1 99.613} C_DIS
LIN {X 0.036,Y -473.722,Z 618.552,A 0.000,B 0.000,C 90.000,E1 99.378} C_DIS
LIN {X 0.022,Y -475.354,Z 618.551,A 0.000,B 0.000,C 90.000,E1 99.151} C_DIS
LIN {X -0.114,Y -476.731,Z 618.549,A 0.000,B 0.000,C 90.000,E1 98.916} C_DIS
LIN {X 0.218,Y -477.752,Z 618.548,A 0.000,B 0.000,C 90.000,E1 98.624} C_DIS
LIN {X -0.115,Y -478.924,Z 618.545,A 0.000,B 0.000,C 90.000,E1 98.163} C_DIS
LIN {X 0.032,Y -479.095,Z 618.542,A 0.000,B 0.000,C 90.000,E1 97.644} C_DIS
LIN {X 0.188,Y -478.290,Z 618.540,A 0.000,B 0.000,C 90.000,E1 97.125} C_DIS
LIN {X -0.129,Y -476.378,Z 618.537,A 0.000,B 0.000,C 90.000,E1 96.663} C_DIS
LIN {X 0.210,Y -474.891,Z 618.536,A 0.000,B 0.000,C 90.000,E1 96.372} C_DIS
LIN {X -0.086,Y -458.879,Z 618.523,A 0.000,B 0.000,C 90.000,E1 94.131} C_DIS
LIN {X -0.080,Y -446.297,Z 618.511,A 0.000,B 0.000,C 90.000,E1 92.064} C_DIS
LIN {X 0.062,Y -434.798,Z 618.500,A 0.000,B 0.000,C 90.000,E1 89.943} C_DIS
LIN {X -0.049,Y -427.366,Z 618.492,A 0.000,B 0.000,C 90.000,E1 88.625} C_DIS
LIN {X -0.143,Y -418.002,Z 618.483,A 0.000,B 0.000,C 90.000,E1 87.020} C_DIS
LIN {X -0.102,Y -403.914,Z 618.470,A 0.000,B 0.000,C 90.000,E1 84.546} C_DIS
LIN {X 0.013,Y -388.896,Z 618.454,A 0.000,B 0.000,C 90.000,E1 81.724} C_DIS
LIN {X -0.095,Y -374.563,Z 618.438,A 0.000,B 0.000,C 90.000,E1 78.870} C_DIS
LIN {X -0.076,Y -362.130,Z 618.423,A 0.000,B 0.000,C 90.000,E1 76.228} C_DIS
LIN {X 0.080,Y -347.839,Z 618.405,A 0.000,B 0.000,C 90.000,E1 72.906} C_DIS
LIN {X 0.144,Y -333.477,Z 618.385,A 0.000,B 0.000,C 90.000,E1 69.209} C_DIS
LIN {X -0.112,Y -320.598,Z 618.364,A 0.000,B 0.000,C 90.000,E1 65.485} C_DIS
LIN {X -0.096,Y -310.873,Z 618.346,A 0.000,B 0.000,C 90.000,E1 62.281} C_DIS
LIN {X -0.009,Y -303.558,Z 618.331,A 0.000,B 0.000,C 90.000,E1 59.665} C_DIS
LIN {X -0.041,Y -294.797,Z 618.313,A 0.000,B 0.000,C 90.000,E1 56.373} C_DIS
LIN {X 0.056,Y -286.650,Z 618.295,A 0.000,B 0.000,C 90.000,E1 53.004} C_DIS
LIN {X 0.116,Y -280.131,Z 618.279,A 0.000,B 0.000,C 90.000,E1 50.275} C_DIS
LIN {X -0.015,Y -274.843,Z 618.268,A 0.000,B 0.000,C 90.000,E1 48.243} C_DIS
LIN {X -0.036,Y -271.049,Z 618.260,A 0.000,B 0.000,C 90.000,E1 46.863} C_DIS
LIN {X -0.114,Y -266.948,Z 618.253,A 0.000,B 0.000,C 90.000,E1 45.486} C_DIS
LIN {X 0.057,Y -260.350,Z 618.241,A 0.000,B 0.000,C 90.000,E1 43.338} C_DIS
LIN {X -0.067,Y -252.408,Z 618.227,A 0.000,B 0.000,C 90.000,E1 40.862} C_DIS
LIN {X 0.021,Y -242.666,Z 618.209,A 0.000,B 0.000,C 90.000,E1 37.569} C_DIS
LIN {X 0.014,Y -234.740,Z 618.192,A 0.000,B 0.000,C 90.000,E1 34.612} C_DIS
LIN {X 0.066,Y -227.604,Z 618.176,A 0.000,B 0.000,C 90.000,E1 31.592} C_DIS
LIN {X -0.022,Y -221.116,Z 618.159,A 0.000,B 0.000,C 90.000,E1 28.565} C_DIS
LIN {X 0.017,Y -215.383,Z 618.141,A 0.000,B 0.000,C 90.000,E1 25.463} C_DIS
LIN {X 0.022,Y -210.414,Z 618.124,A 0.000,B 0.000,C 90.000,E1 22.333} C_DIS
LIN {X 0.075,Y -205.298,Z 618.102,A 0.000,B 0.000,C 90.000,E1 18.362} C_DIS
LIN {X 0.102,Y -201.289,Z 618.080,A 0.000,B 0.000,C 90.000,E1 14.356} C_DIS
LIN {X -0.044,Y -197.848,Z 618.053,A 0.000,B 0.000,C 90.000,E1 9.557} C_DIS
LIN {X -0.033,Y -195.592,Z 618.012,A 0.000,B 0.000,C 90.000,E1 2.236} C_DIS
LIN {X 0.059,Y -197.333,Z 617.961,A 0.000,B 0.000,C 90.000,E1 352.996} C_DIS
LIN {X -0.095,Y -200.295,Z 617.934,A 0.000,B 0.000,C 90.000,E1 348.173} C_DIS
LIN {X 0.056,Y -203.891,Z 617.912,A 0.000,B 0.000,C 90.000,E1 344.102} C_DIS
LIN {X 0.027,Y -208.446,Z 617.890,A 0.000,B 0.000,C 90.000,E1 340.115} C_DIS
LIN {X -0.036,Y -213.724,Z 617.868,A 0.000,B 0.000,C 90.000,E1 336.177} C_DIS
LIN {X -0.091,Y -219.677,Z 617.846,A 0.000,B 0.000,C 90.000,E1 332.281} C_DIS
LIN {X -0.035,Y -226.331,Z 617.824,A 0.000,B 0.000,C 90.000,E1 328.408} C_DIS
LIN {X -0.061,Y -233.589,Z 617.803,A 0.000,B 0.000,C 90.000,E1 324.609} C_DIS
LIN {X -0.007,Y -241.320,Z 617.782,A 0.000,B 0.000,C 90.000,E1 320.848} C_DIS
LIN {X 0.041,Y -249.698,Z 617.762,A 0.000,B 0.000,C 90.000,E1 317.148} C_DIS
LIN {X -0.045,Y -259.046,Z 617.742,A 0.000,B 0.000,C 90.000,E1 313.542} C_DIS
LIN {X -0.013,Y -268.625,Z 617.724,A 0.000,B 0.000,C 90.000,E1 310.334} C_DIS
LIN {X -0.109,Y -280.902,Z 617.705,A 0.000,B 0.000,C 90.000,E1 306.870} C_DIS
LIN {X -0.027,Y -294.685,Z 617.686,A 0.000,B 0.000,C 90.000,E1 303.452} C_DIS
LIN {X -0.014,Y -308.534,Z 617.669,A 0.000,B 0.000,C 90.000,E1 300.463} C_DIS
LIN {X 0.121,Y -321.785,Z 617.655,A 0.000,B 0.000,C 90.000,E1 297.847} C_DIS
LIN {X 0.007,Y -335.560,Z 617.641,A 0.000,B 0.000,C 90.000,E1 295.335} C_DIS
LIN {X -0.115,Y -355.954,Z 617.622,A 0.000,B 0.000,C 90.000,E1 291.972} C_DIS
LIN {X 0.113,Y -376.622,Z 617.605,A 0.000,B 0.000,C 90.000,E1 288.960} C_DIS
LIN {X 0.155,Y -399.551,Z 617.589,A 0.000,B 0.000,C 90.000,E1 286.079} C_DIS
LIN {X -0.091,Y -411.086,Z 617.582,A 0.000,B 0.000,C 90.000,E1 284.717} C_DIS
LIN {X -0.190,Y -422.336,Z 617.574,A 0.000,B 0.000,C 90.000,E1 283.355} C_DIS
LIN {X 0.020,Y -431.088,Z 617.568,A 0.000,B 0.000,C 90.000,E1 282.243} C_DIS
LIN {X 0.116,Y -441.640,Z 617.561,A 0.000,B 0.000,C 90.000,E1 280.894} C_DIS
LIN {X 0.052,Y -449.666,Z 617.555,A 0.000,B 0.000,C 90.000,E1 279.849} C_DIS
LIN {X 0.166,Y -461.181,Z 617.546,A 0.000,B 0.000,C 90.000,E1 278.276} C_DIS
LIN {X -0.198,Y -468.448,Z 617.540,A 0.000,B 0.000,C 90.000,E1 277.296} C_DIS
LIN {X 0.197,Y -473.340,Z 617.536,A 0.000,B 0.000,C 90.000,E1 276.486} C_DIS
LIN {X 0.111,Y -477.471,Z 617.532,A 0.000,B 0.000,C 90.000,E1 275.739} C_DIS
LIN {X -0.226,Y -479.751,Z 617.529,A 0.000,B 0.000,C 90.000,E1 275.277} C_DIS
LIN {X -0.075,Y -481.735,Z 617.526,A 0.000,B 0.000,C 90.000,E1 274.759} C_DIS
LIN {X 0.046,Y -483.297,Z 617.524,A 0.000,B 0.000,C 90.000,E1 274.245} C_DIS
LIN {X 0.217,Y -484.494,Z 617.521,A 0.000,B 0.000,C 90.000,E1 273.726} C_DIS
LIN {X -0.118,Y -485.365,Z 617.518,A 0.000,B 0.000,C 90.000,E1 273.269} C_DIS
LIN {X 0.065,Y -485.912,Z 617.515,A 0.000,B 0.000,C 90.000,E1 272.751} C_DIS
LIN {X 0.229,Y -486.172,Z 617.513,A 0.000,B 0.000,C 90.000,E1 272.236} C_DIS
LIN {X -0.072,Y -486.120,Z 617.510,A 0.000,B 0.000,C 90.000,E1 271.776} C_DIS
LIN {X 0.099,Y -485.679,Z 617.507,A 0.000,B 0.000,C 90.000,E1 271.260} C_DIS
LIN {X -0.216,Y -484.858,Z 617.504,A 0.000,B 0.000,C 90.000,E1 270.802} C_DIS
LIN {X -0.047,Y -483.530,Z 617.502,A 0.000,B 0.000,C 90.000,E1 270.286} C_DIS
LIN {X 0.117,Y -481.608,Z 617.499,A 0.000,B 0.000,C 90.000,E1 269.771} C_DIS
LIN {X -0.207,Y -479.011,Z 617.496,A 0.000,B 0.000,C 90.000,E1 269.312} C_DIS
LIN {X -0.070,Y -475.639,Z 617.493,A 0.000,B 0.000,C 90.000,E1 268.797} C_DIS
LIN {X 0.047,Y -471.310,Z 617.490,A 0.000,B 0.000,C 90.000,E1 268.282} C_DIS
LIN {X 0.155,Y -465.682,Z 617.488,A 0.000,B 0.000,C 90.000,E1 267.764} C_DIS
LIN {X 0.192,Y -462.696,Z 617.486,A 0.000,B 0.000,C 90.000,E1 267.535} C_DIS
LIN {X 0.226,Y -459.232,Z 617.485,A 0.000,B 0.000,C 90.000,E1 267.306} C_DIS
LIN {X 0.128,Y -455.965,Z 617.484,A 0.000,B 0.000,C 90.000,E1 267.135} C_DIS
LIN {X -0.167,Y -448.736,Z 617.482,A 0.000,B 0.000,C 90.000,E1 266.846} C_DIS
LIN {X 0.054,Y -441.362,Z 617.481,A 0.000,B 0.000,C 90.000,E1 266.560} C_DIS
LIN {X -0.176,Y -433.438,Z 617.480,A 0.000,B 0.000,C 90.000,E1 266.388} C_DIS
LIN {X 0.017,Y -424.929,Z 617.479,A 0.000,B 0.000,C 90.000,E1 266.216} C_DIS
LIN {X 0.120,Y -414.192,Z 617.478,A 0.000,B 0.000,C 90.000,E1 266.102} C_DIS
LIN {X 0.047,Y -411.668,Z 617.478,A 0.000,B 0.000,C 90.000,E1 266.102} C_DIS
LIN {X -0.012,Y -180.924,Z 617.478,A 0.000,B 0.000,C 90.000,E1 266.102} C_DIS
LIN {X -0.019,Y -180.899,Z 617.474,A 0.000,B 0.000,C 90.000,E1 265.241} C_DIS
LIN {X -0.069,Y -180.215,Z 617.464,A 0.000,B 0.000,C 90.000,E1 263.571} C_DIS
LIN {X 0.061,Y -179.034,Z 617.445,A 0.000,B 0.000,C 90.000,E1 260.151} C_DIS
LIN {X -0.053,Y -178.692,Z 617.441,A 0.000,B 0.000,C 90.000,E1 259.342} C_DIS
LIN {X 0.057,Y -175.740,Z 617.412,A 0.000,B 0.000,C 90.000,E1 254.212} C_DIS
LIN {X 0.053,Y -171.925,Z 617.384,A 0.000,B 0.000,C 90.000,E1 249.082} C_DIS
LIN {X 0.028,Y -171.298,Z 617.379,A 0.000,B 0.000,C 90.000,E1 248.230} C_DIS
LIN {X 0.073,Y -167.560,Z 617.355,A 0.000,B 0.000,C 90.000,E1 243.896} C_DIS
LIN {X 0.086,Y -166.186,Z 617.345,A 0.000,B 0.000,C 90.000,E1 242.153} C_DIS
LIN {X 0.076,Y -162.955,Z 617.326,A 0.000,B 0.000,C 90.000,E1 238.663} C_DIS
LIN {X -0.100,Y -160.863,Z 617.311,A 0.000,B 0.000,C 90.000,E1 236.087} C_DIS
LIN {X 0.100,Y -157.638,Z 617.292,A 0.000,B 0.000,C 90.000,E1 232.477} C_DIS
LIN {X 0.038,Y -155.676,Z 617.277,A 0.000,B 0.000,C 90.000,E1 229.828} C_DIS
LIN {X -0.017,Y -151.942,Z 617.252,A 0.000,B 0.000,C 90.000,E1 225.364} C_DIS
LIN {X -0.007,Y -150.180,Z 617.237,A 0.000,B 0.000,C 90.000,E1 222.651} C_DIS
LIN {X 0.023,Y -146.955,Z 617.212,A 0.000,B 0.000,C 90.000,E1 218.096} C_DIS
LIN {X 0.011,Y -145.542,Z 617.196,A 0.000,B 0.000,C 90.000,E1 215.358} C_DIS
LIN {X -0.072,Y -142.938,Z 617.171,A 0.000,B 0.000,C 90.000,E1 210.797} C_DIS
LIN {X -0.015,Y -141.562,Z 617.150,A 0.000,B 0.000,C 90.000,E1 207.078} C_DIS
LIN {X 0.037,Y -139.409,Z 617.114,A 0.000,B 0.000,C 90.000,E1 200.556} C_DIS
LIN {X -0.042,Y -139.131,Z 617.104,A 0.000,B 0.000,C 90.000,E1 198.725} C_DIS
LIN {X -0.014,Y -138.350,Z 617.057,A 0.000,B 0.000,C 90.000,E1 190.310} C_DIS
LIN {X -0.026,Y -139.498,Z 617.005,A 0.000,B 0.000,C 90.000,E1 180.974} C_DIS
LIN {X 0.055,Y -141.119,Z 616.974,A 0.000,B 0.000,C 90.000,E1 175.355} C_DIS
LIN {X 0.008,Y -142.499,Z 616.959,A 0.000,B 0.000,C 90.000,E1 172.591} C_DIS
LIN {X -0.046,Y -144.753,Z 616.933,A 0.000,B 0.000,C 90.000,E1 167.993} C_DIS
LIN {X 0.046,Y -147.362,Z 616.913,A 0.000,B 0.000,C 90.000,E1 164.283} C_DIS
LIN {X -0.032,Y -150.689,Z 616.887,A 0.000,B 0.000,C 90.000,E1 159.752} C_DIS
LIN {X 0.051,Y -154.169,Z 616.867,A 0.000,B 0.000,C 90.000,E1 156.102} C_DIS
LIN {X -0.018,Y -157.603,Z 616.847,A 0.000,B 0.000,C 90.000,E1 152.538} C_DIS
LIN {X -0.068,Y -161.855,Z 616.828,A 0.000,B 0.000,C 90.000,E1 148.997} C_DIS
LIN {X -0.050,Y -166.045,Z 616.808,A 0.000,B 0.000,C 90.000,E1 145.468} C_DIS
LIN {X -0.060,Y -171.049,Z 616.789,A 0.000,B 0.000,C 90.000,E1 141.984} C_DIS
LIN {X -0.029,Y -175.920,Z 616.770,A 0.000,B 0.000,C 90.000,E1 138.528} C_DIS
LIN {X -0.037,Y -180.159,Z 616.755,A 0.000,B 0.000,C 90.000,E1 135.972} C_DIS
LIN {X -0.069,Y -185.576,Z 616.737,A 0.000,B 0.000,C 90.000,E1 132.609} C_DIS
LIN {X 0.027,Y -191.174,Z 616.720,A 0.000,B 0.000,C 90.000,E1 129.519} C_DIS
LIN {X -0.005,Y -288.619,Z 616.720,A 0.000,B 0.000,C 90.000,E1 129.519} C_DIS
LIN {X 0.043,Y -290.205,Z 616.719,A 0.000,B 0.000,C 90.000,E1 129.483} C_DIS
LIN {X -0.101,Y -294.961,Z 616.718,A 0.000,B 0.000,C 90.000,E1 129.277} C_DIS
LIN {X -0.012,Y -298.176,Z 616.716,A 0.000,B 0.000,C 90.000,E1 128.955} C_DIS
LIN {X 0.136,Y -301.821,Z 616.713,A 0.000,B 0.000,C 90.000,E1 128.382} C_DIS
LIN {X -0.106,Y -303.377,Z 616.712,A 0.000,B 0.000,C 90.000,E1 128.096} C_DIS
LIN {X 0.080,Y -304.601,Z 616.710,A 0.000,B 0.000,C 90.000,E1 127.729} C_DIS
LIN {X -0.028,Y -316.238,Z 616.688,A 0.000,B 0.000,C 90.000,E1 123.833} C_DIS
LIN {X 0.140,Y -326.340,Z 616.672,A 0.000,B 0.000,C 90.000,E1 120.924} C_DIS
LIN {X 0.108,Y -337.778,Z 616.656,A 0.000,B 0.000,C 90.000,E1 118.103} C_DIS
LIN {X 0.091,Y -350.647,Z 616.641,A 0.000,B 0.000,C 90.000,E1 115.335} C_DIS
LIN {X -0.083,Y -363.387,Z 616.627,A 0.000,B 0.000,C 90.000,E1 112.950} C_DIS
LIN {X 0.127,Y -377.444,Z 616.614,A 0.000,B 0.000,C 90.000,E1 110.556} C_DIS
LIN {X 0.213,Y -392.919,Z 616.602,A 0.000,B 0.000,C 90.000,E1 108.236} C_DIS
LIN {X -0.069,Y -409.926,Z 616.589,A 0.000,B 0.000,C 90.000,E1 106.024} C_DIS
LIN {X -0.052,Y -428.590,Z 616.577,A 0.000,B 0.000,C 90.000,E1 103.828} C_DIS
LIN {X 0.172,Y -448.556,Z 616.565,A 0.000,B 0.000,C 90.000,E1 101.715} C_DIS
LIN {X -0.202,Y -469.104,Z 616.555,A 0.000,B 0.000,C 90.000,E1 99.849} C_DIS
LIN {X -0.148,Y -471.710,Z 616.553,A 0.000,B 0.000,C 90.000,E1 99.613} C_DIS
LIN {X -0.086,Y -473.849,Z 616.552,A 0.000,B 0.000,C 90.000,E1 99.378} C_DIS
LIN {X -0.101,Y -475.475,Z 616.551,A 0.000,B 0.000,C 90.000,E1 99.151} C_DIS
LIN {X 0.233,Y -476.845,Z 616.549,A 0.000,B 0.000,C 90.000,E1 98.859} C_DIS
LIN {X 0.094,Y -477.861,Z 616.548,A 0.000,B 0.000,C 90.000,E1 98.624} C_DIS
LIN {X 0.235,Y -479.026,Z 616.545,A 0.000,B 0.000,C 90.000,E1 98.106} C_DIS
LIN {X -0.090,Y -479.188,Z 616.542,A 0.000,B 0.000,C 90.000,E1 97.644} C_DIS
LIN {X 0.066,Y -478.376,Z 616.540,A 0.000,B 0.000,C 90.000,E1 97.125} C_DIS
LIN {X -0.250,Y -476.455,Z 616.537,A 0.000,B 0.000,C 90.000,E1 96.663} C_DIS
LIN {X 0.089,Y -474.960,Z 616.535,A 0.000,B 0.000,C 90.000,E1 96.372} C_DIS
LIN {X -0.200,Y -458.925,Z 616.523,A 0.000,B 0.000,C 90.000,E1 94.131} C_DIS
LIN {X -0.191,Y -446.331,Z 616.511,A 0.000,B 0.000,C 90.000,E1 92.064} C_DIS
LIN {X -0.045,Y -434.810,Z 616.500,A 0.000,B 0.000,C 90.000,E1 89.943} C_DIS
LIN {X -0.154,Y -427.380,Z 616.492,A 0.000,B 0.000,C 90.000,E1 88.625} C_DIS
LIN {X 0.172,Y -418.014,Z 616.483,A 0.000,B 0.000,C 90.000,E1 86.963} C_DIS
LIN {X 0.202,Y -403.909,Z 616.470,A 0.000,B 0.000,C 90.000,E1 84.489} C_DIS
LIN {X -0.082,Y -388.899,Z 616.454,A 0.000,B 0.000,C 90.000,E1 81.724} C_DIS
LIN {X 0.165,Y -375.968,Z 616.440,A 0.000,B 0.000,C 90.000,E1 79.106} C_DIS
LIN {X -0.138,Y -363.487,Z 616.425,A 0.000,B 0.000,C 90.000,E1 76.520} C_DIS
LIN {X 0.067,Y -349.091,Z 616.407,A 0.000,B 0.000,C 90.000,E1 73.196} C_DIS
LIN {X 0.073,Y -334.636,Z 616.386,A 0.000,B 0.000,C 90.000,E1 69.518} C_DIS
LIN {X -0.096,Y -322.673,Z 616.367,A 0.000,B 0.000,C 90.000,E1 66.102} C_DIS
LIN {X 0.129,Y -312.849,Z 616.349,A 0.000,B 0.000,C 90.000,E1 62.871} C_DIS
LIN {X -0.078,Y -303.641,Z 616.331,A 0.000,B 0.000,C 90.000,E1 59.665} C_DIS
LIN {X 0.057,Y -294.870,Z 616.313,A 0.000,B 0.000,C 90.000,E1 56.342} C_DIS
LIN {X -0.005,Y -286.711,Z 616.294,A 0.000,B 0.000,C 90.000,E1 53.004} C_DIS
LIN {X 0.023,Y -281.815,Z 616.283,A 0.000,B 0.000,C 90.000,E1 50.964} C_DIS
LIN {X -0.095,Y -278.477,Z 616.276,A 0.000,B 0.000,C 90.000,E1 49.622} C_DIS
LIN {X -0.075,Y -273.036,Z 616.264,A 0.000,B 0.000,C 90.000,E1 47.553} C_DIS
LIN {X 0.066,Y -269.085,Z 616.256,A 0.000,B 0.000,C 90.000,E1 46.134} C_DIS
LIN {X 0.083,Y -262.650,Z 616.245,A 0.000,B 0.000,C 90.000,E1 44.028} C_DIS
LIN {X -0.023,Y -255.836,Z 616.233,A 0.000,B 0.000,C 90.000,E1 41.919} C_DIS
LIN {X -0.024,Y -244.797,Z 616.213,A 0.000,B 0.000,C 90.000,E1 38.302} C_DIS
LIN {X -0.032,Y -236.679,Z 616.196,A 0.000,B 0.000,C 90.000,E1 35.358} C_DIS
LIN {X 0.066,Y -229.352,Z 616.180,A 0.000,B 0.000,C 90.000,E1 32.339} C_DIS
LIN {X -0.055,Y -221.140,Z 616.159,A 0.000,B 0.000,C 90.000,E1 28.565} C_DIS
LIN {X -0.015,Y -215.404,Z 616.141,A 0.000,B 0.000,C 90.000,E1 25.463} C_DIS
LIN {X -0.009,Y -210.416,Z 616.124,A 0.000,B 0.000,C 90.000,E1 22.333} C_DIS
LIN {X 0.045,Y -205.308,Z 616.102,A 0.000,B 0.000,C 90.000,E1 18.362} C_DIS
LIN {X 0.074,Y -201.315,Z 616.080,A 0.000,B 0.000,C 90.000,E1 14.356} C_DIS
LIN {X -0.072,Y -197.871,Z 616.053,A 0.000,B 0.000,C 90.000,E1 9.557} C_DIS
LIN {X -0.060,Y -195.610,Z 616.012,A 0.000,B 0.000,C 90.000,E1 2.236} C_DIS
LIN {X 0.061,Y -197.373,Z 615.961,A 0.000,B 0.000,C 90.000,E1 352.996} C_DIS
LIN {X -0.091,Y -200.368,Z 615.934,A 0.000,B 0.000,C 90.000,E1 348.173} C_DIS
LIN {X 0.061,Y -203.952,Z 615.912,A 0.000,B 0.000,C 90.000,E1 344.102} C_DIS
LIN {X -0.026,Y -209.501,Z 615.885,A 0.000,B 0.000,C 90.000,E1 339.337} C_DIS
LIN {X 0.102,Y -214.907,Z 615.863,A 0.000,B 0.000,C 90.000,E1 335.357} C_DIS
LIN {X -0.109,Y -220.964,Z 615.842,A 0.000,B 0.000,C 90.000,E1 331.513} C_DIS
LIN {X -0.097,Y -227.762,Z 615.820,A 0.000,B 0.000,C 90.000,E1 327.661} C_DIS
LIN {X -0.048,Y -233.611,Z 615.803,A 0.000,B 0.000,C 90.000,E1 324.609} C_DIS
LIN {X 0.007,Y -241.324,Z 615.782,A 0.000,B 0.000,C 90.000,E1 320.848} C_DIS
LIN {X 0.055,Y -249.678,Z 615.762,A 0.000,B 0.000,C 90.000,E1 317.148} C_DIS
LIN {X -0.032,Y -258.991,Z 615.742,A 0.000,B 0.000,C 90.000,E1 313.542} C_DIS
LIN {X 0.000,Y -268.563,Z 615.724,A 0.000,B 0.000,C 90.000,E1 310.334} C_DIS
LIN {X -0.098,Y -280.813,Z 615.705,A 0.000,B 0.000,C 90.000,E1 306.870} C_DIS
LIN {X -0.018,Y -294.575,Z 615.686,A 0.000,B 0.000,C 90.000,E1 303.452} C_DIS
LIN {X -0.008,Y -308.466,Z 615.669,A 0.000,B 0.000,C 90.000,E1 300.463} C_DIS
LIN {X -0.080,Y -323.372,Z 615.653,A 0.000,B 0.000,C 90.000,E1 297.564} C_DIS
LIN {X 0.094,Y -340.825,Z 615.636,A 0.000,B 0.000,C 90.000,E1 294.387} C_DIS
LIN {X -0.080,Y -357.858,Z 615.620,A 0.000,B 0.000,C 90.000,E1 291.663} C_DIS
LIN {X 0.108,Y -376.566,Z 615.605,A 0.000,B 0.000,C 90.000,E1 288.960} C_DIS
LIN {X 0.148,Y -399.528,Z 615.589,A 0.000,B 0.000,C 90.000,E1 286.079} C_DIS
LIN {X -0.123,Y -411.093,Z 615.582,A 0.000,B 0.000,C 90.000,E1 284.717} C_DIS
LIN {X 0.186,Y -422.369,Z 615.574,A 0.000,B 0.000,C 90.000,E1 283.300} C_DIS
LIN {X 0.158,Y -433.263,Z 615.567,A 0.000,B 0.000,C 90.000,E1 281.951} C_DIS
LIN {X -0.139,Y -443.708,Z 615.559,A 0.000,B 0.000,C 90.000,E1 280.658} C_DIS
LIN {X -0.185,Y -451.658,Z 615.553,A 0.000,B 0.000,C 90.000,E1 279.613} C_DIS
LIN {X -0.113,Y -463.028,Z 615.545,A 0.000,B 0.000,C 90.000,E1 278.049} C_DIS
LIN {X 0.068,Y -470.069,Z 615.539,A 0.000,B 0.000,C 90.000,E1 277.004} C_DIS
LIN {X -0.050,Y -474.673,Z 615.535,A 0.000,B 0.000,C 90.000,E1 276.258} C_DIS
LIN {X -0.119,Y -478.562,Z 615.531,A 0.000,B 0.000,C 90.000,E1 275.511} C_DIS
LIN {X -0.114,Y -481.648,Z 615.526,A 0.000,B 0.000,C 90.000,E1 274.759} C_DIS
LIN {X 0.006,Y -483.200,Z 615.524,A 0.000,B 0.000,C 90.000,E1 274.245} C_DIS
LIN {X 0.176,Y -484.441,Z 615.521,A 0.000,B 0.000,C 90.000,E1 273.726} C_DIS
LIN {X -0.160,Y -485.307,Z 615.518,A 0.000,B 0.000,C 90.000,E1 273.269} C_DIS
LIN {X 0.023,Y -485.872,Z 615.515,A 0.000,B 0.000,C 90.000,E1 272.751} C_DIS
LIN {X 0.187,Y -486.140,Z 615.513,A 0.000,B 0.000,C 90.000,E1 272.236} C_DIS
LIN {X -0.114,Y -486.123,Z 615.510,A 0.000,B 0.000,C 90.000,E1 271.776} C_DIS
LIN {X 0.056,Y -485.709,Z 615.507,A 0.000,B 0.000,C 90.000,E1 271.260} C_DIS
LIN {X 0.227,Y -484.912,Z 615.504,A 0.000,B 0.000,C 90.000,E1 270.745} C_DIS
LIN {X -0.089,Y -483.564,Z 615.502,A 0.000,B 0.000,C 90.000,E1 270.286} C_DIS
LIN {X 0.076,Y -481.637,Z 615.499,A 0.000,B 0.000,C 90.000,E1 269.771} C_DIS
LIN {X 0.231,Y -479.029,Z 615.496,A 0.000,B 0.000,C 90.000,E1 269.255} C_DIS
LIN {X -0.111,Y -475.645,Z 615.493,A 0.000,B 0.000,C 90.000,E1 268.797} C_DIS
LIN {X 0.006,Y -471.279,Z 615.490,A 0.000,B 0.000,C 90.000,E1 268.282} C_DIS
LIN {X -0.166,Y -468.665,Z 615.489,A 0.000,B 0.000,C 90.000,E1 268.051} C_DIS
LIN {X 0.193,Y -462.745,Z 615.486,A 0.000,B 0.000,C 90.000,E1 267.535} C_DIS
LIN {X 0.193,Y -456.093,Z 615.484,A 0.000,B 0.000,C 90.000,E1 267.135} C_DIS
LIN {X -0.098,Y -448.906,Z 615.482,A 0.000,B 0.000,C 90.000,E1 266.846} C_DIS
LIN {X 0.100,Y -441.564,Z 615.481,A 0.000,B 0.000,C 90.000,E1 266.560} C_DIS
LIN {X -0.134,Y -433.760,Z 615.480,A 0.000,B 0.000,C 90.000,E1 266.388} C_DIS
LIN {X 0.046,Y -425.336,Z 615.479,A 0.000,B 0.000,C 90.000,E1 266.216} C_DIS
LIN {X 0.063,Y -412.963,Z 615.478,A 0.000,B 0.000,C 90.000,E1 266.102} C_DIS
LIN {X -0.010,Y -405.007,Z 615.478,A 0.000,B 0.000,C 90.000,E1 266.102} C_DIS
LIN {X -0.037,Y -180.924,Z 615.478,A 0.000,B 0.000,C 90.000,E1 266.102} C_DIS
LIN {X 0.007,Y -180.876,Z 615.473,A 0.000,B 0.000,C 90.000,E1 265.065} C_DIS
LIN {X 0.089,Y -178.942,Z 615.443,A 0.000,B 0.000,C 90.000,E1 259.803} C_DIS
LIN {X -0.044,Y -175.993,Z 615.415,A 0.000,B 0.000,C 90.000,E1 254.755} C_DIS
LIN {X -0.098,Y -175.495,Z 615.411,A 0.000,B 0.000,C 90.000,E1 253.921} C_DIS
LIN {X -0.034,Y -172.238,Z 615.387,A 0.000,B 0.000,C 90.000,E1 249.625} C_DIS
LIN {X -0.055,Y -171.716,Z 615.382,A 0.000,B 0.000,C 90.000,E1 248.773} C_DIS
LIN {X -0.046,Y -167.311,Z 615.353,A 0.000,B 0.000,C 90.000,E1 243.589} C_DIS
LIN {X 0.034,Y -166.692,Z 615.348,A 0.000,B 0.000,C 90.000,E1 242.692} C_DIS
LIN {X 0.025,Y -162.673,Z 615.324,A 0.000,B 0.000,C 90.000,E1 238.329} C_DIS
LIN {X -0.002,Y -161.364,Z 615.314,A 0.000,B 0.000,C 90.000,E1 236.580} C_DIS
LIN {X 0.032,Y -157.357,Z 615.290,A 0.000,B 0.000,C 90.000,E1 232.145} C_DIS
LIN {X 0.060,Y -155.346,Z 615.275,A 0.000,B 0.000,C 90.000,E1 229.461} C_DIS
LIN {X -0.010,Y -151.693,Z 615.250,A 0.000,B 0.000,C 90.000,E1 225.000} C_DIS
LIN {X 0.038,Y -150.554,Z 615.240,A 0.000,B 0.000,C 90.000,E1 223.176} C_DIS
LIN {X -0.045,Y -147.281,Z 615.215,A 0.000,B 0.000,C 90.000,E1 218.669} C_DIS
LIN {X -0.076,Y -145.309,Z 615.194,A 0.000,B 0.000,C 90.000,E1 215.025} C_DIS
LIN {X 0.034,Y -142.400,Z 615.164,A 0.000,B 0.000,C 90.000,E1 209.461} C_DIS
LIN {X 0.017,Y -141.382,Z 615.148,A 0.000,B 0.000,C 90.000,E1 206.693} C_DIS
LIN {X 0.058,Y -139.349,Z 615.112,A 0.000,B 0.000,C 90.000,E1 200.174} C_DIS
LIN {X 0.000,Y -138.786,Z 615.097,A 0.000,B 0.000,C 90.000,E1 197.402} C_DIS
LIN {X 0.058,Y -138.344,Z 615.055,A 0.000,B 0.000,C 90.000,E1 189.905} C_DIS
LIN {X -0.061,Y -139.386,Z 615.008,A 0.000,B 0.000,C 90.000,E1 181.547} C_DIS
LIN {X -0.008,Y -141.283,Z 614.972,A 0.000,B 0.000,C 90.000,E1 175.008} C_DIS
LIN {X -0.050,Y -142.646,Z 614.957,A 0.000,B 0.000,C 90.000,E1 172.243} C_DIS
LIN {X 0.042,Y -144.982,Z 614.931,A 0.000,B 0.000,C 90.000,E1 167.589} C_DIS
LIN {X 0.032,Y -147.610,Z 614.911,A 0.000,B 0.000,C 90.000,E1 163.921} C_DIS
LIN {X -0.031,Y -150.232,Z 614.890,A 0.000,B 0.000,C 90.000,E1 160.296} C_DIS
LIN {X -0.015,Y -153.622,Z 614.870,A 0.000,B 0.000,C 90.000,E1 156.666} C_DIS
LIN {X -0.027,Y -157.039,Z 614.850,A 0.000,B 0.000,C 90.000,E1 153.076} C_DIS
LIN {X -0.096,Y -161.164,Z 614.831,A 0.000,B 0.000,C 90.000,E1 149.537} C_DIS
LIN {X -0.014,Y -163.259,Z 614.821,A 0.000,B 0.000,C 90.000,E1 147.740} C_DIS
LIN {X 0.085,Y -167.699,Z 614.801,A 0.000,B 0.000,C 90.000,E1 144.196} C_DIS
LIN {X -0.002,Y -171.519,Z 614.787,A 0.000,B 0.000,C 90.000,E1 141.618} C_DIS
LIN {X 0.041,Y -176.456,Z 614.768,A 0.000,B 0.000,C 90.000,E1 138.162} C_DIS
LIN {X -0.089,Y -180.753,Z 614.753,A 0.000,B 0.000,C 90.000,E1 135.648} C_DIS
LIN {X 0.029,Y -186.158,Z 614.735,A 0.000,B 0.000,C 90.000,E1 132.243} C_DIS
LIN {X -0.016,Y -191.194,Z 614.720,A 0.000,B 0.000,C 90.000,E1 129.519} C_DIS
LIN {X 0.110,Y -288.874,Z 614.719,A 0.000,B 0.000,C 90.000,E1 129.483} C_DIS
LIN {X -0.037,Y -290.399,Z 614.719,A 0.000,B 0.000,C 90.000,E1 129.483} C_DIS
LIN {X 0.022,Y -295.557,Z 614.718,A 0.000,B 0.000,C 90.000,E1 129.197} C_DIS
LIN {X 0.082,Y -298.319,Z 614.716,A 0.000,B 0.000,C 90.000,E1 128.910} C_DIS
LIN {X -0.117,Y -302.021,Z 614.713,A 0.000,B 0.000,C 90.000,E1 128.382} C_DIS
LIN {X 0.068,Y -303.537,Z 614.711,A 0.000,B 0.000,C 90.000,E1 128.016} C_DIS
LIN {X 0.068,Y -304.729,Z 614.709,A 0.000,B 0.000,C 90.000,E1 127.684} C_DIS
LIN {X -0.081,Y -315.322,Z 614.689,A 0.000,B 0.000,C 90.000,E1 124.119} C_DIS
LIN {X 0.060,Y -325.304,Z 614.673,A 0.000,B 0.000,C 90.000,E1 121.209} C_DIS
LIN {X 0.169,Y -336.608,Z 614.658,A 0.000,B 0.000,C 90.000,E1 118.359} C_DIS
LIN {X 0.115,Y -349.339,Z 614.642,A 0.000,B 0.000,C 90.000,E1 115.591} C_DIS
LIN {X -0.088,Y -361.944,Z 614.629,A 0.000,B 0.000,C 90.000,E1 113.206} C_DIS
LIN {X -0.130,Y -375.856,Z 614.616,A 0.000,B 0.000,C 90.000,E1 110.844} C_DIS
LIN {X 0.141,Y -391.175,Z 614.603,A 0.000,B 0.000,C 90.000,E1 108.489} C_DIS
LIN {X -0.062,Y -408.013,Z 614.590,A 0.000,B 0.000,C 90.000,E1 106.260} C_DIS
LIN {X -0.095,Y -426.494,Z 614.578,A 0.000,B 0.000,C 90.000,E1 104.064} C_DIS
LIN {X -0.015,Y -446.384,Z 614.566,A 0.000,B 0.000,C 90.000,E1 101.951} C_DIS
LIN {X 0.005,Y -466.874,Z 614.556,A 0.000,B 0.000,C 90.000,E1 100.018} C_DIS
LIN {X 0.041,Y -472.048,Z 614.553,A 0.000,B 0.000,C 90.000,E1 99.557} C_DIS
LIN {X 0.098,Y -474.133,Z 614.552,A 0.000,B 0.000,C 90.000,E1 99.321} C_DIS
LIN {X 0.078,Y -475.721,Z 614.551,A 0.000,B 0.000,C 90.000,E1 99.095} C_DIS
LIN {X -0.057,Y -477.055,Z 614.549,A 0.000,B 0.000,C 90.000,E1 98.859} C_DIS
LIN {X -0.196,Y -478.041,Z 614.548,A 0.000,B 0.000,C 90.000,E1 98.624} C_DIS
LIN {X -0.054,Y -479.155,Z 614.545,A 0.000,B 0.000,C 90.000,E1 98.106} C_DIS
LIN {X 0.096,Y -479.272,Z 614.542,A 0.000,B 0.000,C 90.000,E1 97.587} C_DIS
LIN {X -0.221,Y -478.411,Z 614.539,A 0.000,B 0.000,C 90.000,E1 97.125} C_DIS
LIN {X -0.062,Y -476.430,Z 614.537,A 0.000,B 0.000,C 90.000,E1 96.606} C_DIS
LIN {X -0.195,Y -474.895,Z 614.535,A 0.000,B 0.000,C 90.000,E1 96.372} C_DIS
LIN {X -0.020,Y -458.835,Z 614.523,A 0.000,B 0.000,C 90.000,E1 94.073} C_DIS
LIN {X -0.017,Y -446.244,Z 614.511,A 0.000,B 0.000,C 90.000,E1 92.007} C_DIS
LIN {X 0.123,Y -434.701,Z 614.499,A 0.000,B 0.000,C 90.000,E1 89.885} C_DIS
LIN {X 0.009,Y -427.269,Z 614.492,A 0.000,B 0.000,C 90.000,E1 88.568} C_DIS
LIN {X -0.088,Y -417.893,Z 614.483,A 0.000,B 0.000,C 90.000,E1 86.963} C_DIS
LIN {X -0.053,Y -403.781,Z 614.469,A 0.000,B 0.000,C 90.000,E1 84.489} C_DIS
LIN {X 0.111,Y -388.803,Z 614.454,A 0.000,B 0.000,C 90.000,E1 81.659} C_DIS
LIN {X -0.060,Y -374.463,Z 614.438,A 0.000,B 0.000,C 90.000,E1 78.814} C_DIS
LIN {X -0.049,Y -362.020,Z 614.423,A 0.000,B 0.000,C 90.000,E1 76.172} C_DIS
LIN {X 0.096,Y -347.723,Z 614.405,A 0.000,B 0.000,C 90.000,E1 72.851} C_DIS
LIN {X -0.153,Y -334.563,Z 614.386,A 0.000,B 0.000,C 90.000,E1 69.518} C_DIS
LIN {X -0.021,Y -322.654,Z 614.367,A 0.000,B 0.000,C 90.000,E1 66.049} C_DIS
LIN {X -0.085,Y -312.847,Z 614.349,A 0.000,B 0.000,C 90.000,E1 62.871} C_DIS
LIN {X -0.024,Y -303.649,Z 614.331,A 0.000,B 0.000,C 90.000,E1 59.616} C_DIS
LIN {X 0.101,Y -294.877,Z 614.313,A 0.000,B 0.000,C 90.000,E1 56.294} C_DIS
LIN {X 0.075,Y -288.321,Z 614.298,A 0.000,B 0.000,C 90.000,E1 53.623} C_DIS
LIN {X -0.038,Y -283.446,Z 614.287,A 0.000,B 0.000,C 90.000,E1 51.618} C_DIS
LIN {X 0.107,Y -278.448,Z 614.275,A 0.000,B 0.000,C 90.000,E1 49.542} C_DIS
LIN {X 0.124,Y -273.005,Z 614.264,A 0.000,B 0.000,C 90.000,E1 47.472} C_DIS
LIN {X -0.118,Y -269.054,Z 614.256,A 0.000,B 0.000,C 90.000,E1 46.134} C_DIS
LIN {X -0.098,Y -262.609,Z 614.245,A 0.000,B 0.000,C 90.000,E1 44.028} C_DIS
LIN {X 0.004,Y -254.642,Z 614.231,A 0.000,B 0.000,C 90.000,E1 41.515} C_DIS
LIN {X -0.010,Y -244.737,Z 614.213,A 0.000,B 0.000,C 90.000,E1 38.257} C_DIS
LIN {X -0.012,Y -236.601,Z 614.196,A 0.000,B 0.000,C 90.000,E1 35.311} C_DIS
LIN {X -0.103,Y -229.292,Z 614.180,A 0.000,B 0.000,C 90.000,E1 32.339} C_DIS
LIN {X -0.034,Y -222.660,Z 614.163,A 0.000,B 0.000,C 90.000,E1 29.283} C_DIS
LIN {X 0.046,Y -216.700,Z 614.146,A 0.000,B 0.000,C 90.000,E1 26.181} C_DIS
LIN {X 0.026,Y -210.370,Z 614.124,A 0.000,B 0.000,C 90.000,E1 22.280} C_DIS
LIN {X -0.113,Y -205.277,Z 614.102,A 0.000,B 0.000,C 90.000,E1 18.362} C_DIS
LIN {X -0.081,Y -201.303,Z 614.080,A 0.000,B 0.000,C 90.000,E1 14.356} C_DIS
LIN {X -0.029,Y -197.865,Z 614.053,A 0.000,B 0.000,C 90.000,E1 9.500} C_DIS
LIN {X -0.054,Y -195.565,Z 614.008,A 0.000,B 0.000,C 90.000,E1 1.375} C_DIS
LIN {X 0.061,Y -197.410,Z 613.961,A 0.000,B 0.000,C 90.000,E1 352.996} C_DIS
LIN {X -0.089,Y -200.433,Z 613.934,A 0.000,B 0.000,C 90.000,E1 348.173} C_DIS
LIN {X 0.066,Y -204.017,Z 613.912,A 0.000,B 0.000,C 90.000,E1 344.102} C_DIS
LIN {X 0.040,Y -208.554,Z 613.890,A 0.000,B 0.000,C 90.000,E1 340.115} C_DIS
LIN {X -0.020,Y -213.804,Z 613.868,A 0.000,B 0.000,C 90.000,E1 336.177} C_DIS
LIN {X -0.070,Y -219.739,Z 613.846,A 0.000,B 0.000,C 90.000,E1 332.281} C_DIS
LIN {X -0.012,Y -226.395,Z 613.824,A 0.000,B 0.000,C 90.000,E1 328.408} C_DIS
LIN {X -0.036,Y -233.627,Z 613.803,A 0.000,B 0.000,C 90.000,E1 324.609} C_DIS
LIN {X -0.133,Y -241.325,Z 613.783,A 0.000,B 0.000,C 90.000,E1 320.884} C_DIS
LIN {X 0.068,Y -249.648,Z 613.762,A 0.000,B 0.000,C 90.000,E1 317.148} C_DIS
LIN {X -0.020,Y -258.939,Z 613.742,A 0.000,B 0.000,C 90.000,E1 313.542} C_DIS
LIN {X 0.010,Y -268.508,Z 613.724,A 0.000,B 0.000,C 90.000,E1 310.334} C_DIS
LIN {X -0.089,Y -280.740,Z 613.705,A 0.000,B 0.000,C 90.000,E1 306.870} C_DIS
LIN {X 0.000,Y -293.000,Z 613.688,A 0.000,B 0.000,C 90.000,E1 303.785} C_DIS
LIN {X -0.004,Y -308.395,Z 613.669,A 0.000,B 0.000,C 90.000,E1 300.463} C_DIS
LIN {X 0.128,Y -321.573,Z 613.655,A 0.000,B 0.000,C 90.000,E1 297.847} C_DIS
LIN {X 0.008,Y -335.333,Z 613.641,A 0.000,B 0.000,C 90.000,E1 295.335} C_DIS
LIN {X -0.121,Y -355.776,Z 613.622,A 0.000,B 0.000,C 90.000,E1 291.972} C_DIS
LIN {X -0.001,Y -374.348,Z 613.607,A 0.000,B 0.000,C 90.000,E1 289.268} C_DIS
LIN {X 0.139,Y -399.501,Z 613.589,A 0.000,B 0.000,C 90.000,E1 286.079} C_DIS
LIN {X -0.133,Y -411.084,Z 613.582,A 0.000,B 0.000,C 90.000,E1 284.717} C_DIS
LIN {X -0.093,Y -424.610,Z 613.573,A 0.000,B 0.000,C 90.000,E1 283.063} C_DIS
LIN {X 0.148,Y -433.286,Z 613.567,A 0.000,B 0.000,C 90.000,E1 281.951} C_DIS
LIN {X -0.150,Y -443.762,Z 613.559,A 0.000,B 0.000,C 90.000,E1 280.658} C_DIS
LIN {X -0.195,Y -451.710,Z 613.553,A 0.000,B 0.000,C 90.000,E1 279.613} C_DIS
LIN {X 0.122,Y -461.181,Z 613.546,A 0.000,B 0.000,C 90.000,E1 278.276} C_DIS
LIN {X 0.221,Y -468.268,Z 613.540,A 0.000,B 0.000,C 90.000,E1 277.239} C_DIS
LIN {X 0.150,Y -473.094,Z 613.536,A 0.000,B 0.000,C 90.000,E1 276.486} C_DIS
LIN {X 0.061,Y -477.247,Z 613.532,A 0.000,B 0.000,C 90.000,E1 275.739} C_DIS
LIN {X 0.199,Y -479.592,Z 613.529,A 0.000,B 0.000,C 90.000,E1 275.220} C_DIS
LIN {X -0.128,Y -481.562,Z 613.526,A 0.000,B 0.000,C 90.000,E1 274.759} C_DIS
LIN {X -0.008,Y -483.158,Z 613.524,A 0.000,B 0.000,C 90.000,E1 274.245} C_DIS
LIN {X 0.162,Y -484.388,Z 613.521,A 0.000,B 0.000,C 90.000,E1 273.726} C_DIS
LIN {X -0.175,Y -485.270,Z 613.518,A 0.000,B 0.000,C 90.000,E1 273.269} C_DIS
LIN {X 0.007,Y -485.840,Z 613.515,A 0.000,B 0.000,C 90.000,E1 272.751} C_DIS
LIN {X 0.172,Y -486.130,Z 613.513,A 0.000,B 0.000,C 90.000,E1 272.236} C_DIS
LIN {X -0.129,Y -486.138,Z 613.510,A 0.000,B 0.000,C 90.000,E1 271.776} C_DIS
LIN {X 0.040,Y -485.768,Z 613.507,A 0.000,B 0.000,C 90.000,E1 271.260} C_DIS
LIN {X 0.211,Y -484.937,Z 613.504,A 0.000,B 0.000,C 90.000,E1 270.745} C_DIS
LIN {X -0.104,Y -483.596,Z 613.502,A 0.000,B 0.000,C 90.000,E1 270.286} C_DIS
LIN {X 0.061,Y -481.694,Z 613.499,A 0.000,B 0.000,C 90.000,E1 269.771} C_DIS
LIN {X 0.216,Y -479.065,Z 613.496,A 0.000,B 0.000,C 90.000,E1 269.255} C_DIS
LIN {X -0.125,Y -475.658,Z 613.493,A 0.000,B 0.000,C 90.000,E1 268.797} C_DIS
LIN {X 0.171,Y -473.625,Z 613.492,A 0.000,B 0.000,C 90.000,E1 268.511} C_DIS
LIN {X -0.180,Y -468.663,Z 613.489,A 0.000,B 0.000,C 90.000,E1 268.051} C_DIS
LIN {X 0.102,Y -465.686,Z 613.488,A 0.000,B 0.000,C 90.000,E1 267.764} C_DIS
LIN {X 0.152,Y -462.635,Z 613.486,A 0.000,B 0.000,C 90.000,E1 267.535} C_DIS
LIN {X 0.200,Y -459.148,Z 613.485,A 0.000,B 0.000,C 90.000,E1 267.306} C_DIS
LIN {X 0.118,Y -455.891,Z 613.484,A 0.000,B 0.000,C 90.000,E1 267.135} C_DIS
LIN {X -0.172,Y -448.660,Z 613.482,A 0.000,B 0.000,C 90.000,E1 266.846} C_DIS
LIN {X 0.036,Y -441.350,Z 613.481,A 0.000,B 0.000,C 90.000,E1 266.560} C_DIS
LIN {X -0.175,Y -433.491,Z 613.480,A 0.000,B 0.000,C 90.000,E1 266.388} C_DIS
LIN {X 0.030,Y -424.962,Z 613.479,A 0.000,B 0.000,C 90.000,E1 266.216} C_DIS
LIN {X 0.044,Y -412.456,Z 613.478,A 0.000,B 0.000,C 90.000,E1 266.102} C_DIS
LIN {X -0.013,Y -180.924,Z 613.478,A 0.000,B 0.000,C 90.000,E1 266.102} C_DIS
LIN {X -0.021,Y -180.899,Z 613.474,A 0.000,B 0.000,C 90.000,E1 265.241} C_DIS
LIN {X -0.071,Y -180.214,Z 613.464,A 0.000,B 0.000,C 90.000,E1 263.571} C_DIS
LIN {X 0.059,Y -179.033,Z 613.445,A 0.000,B 0.000,C 90.000,E1 260.151} C_DIS
LIN {X -0.055,Y -178.691,Z 613.441,A 0.000,B 0.000,C 90.000,E1 259.342} C_DIS
LIN {X 0.056,Y -175.740,Z 613.412,A 0.000,B 0.000,C 90.000,E1 254.212} C_DIS
LIN {X 0.051,Y -171.924,Z 613.384,A 0.000,B 0.000,C 90.000,E1 249.082} C_DIS
LIN {X 0.026,Y -171.298,Z 613.379,A 0.000,B 0.000,C 90.000,E1 248.230} C_DIS
LIN {X 0.072,Y -167.560,Z 613.355,A 0.000,B 0.000,C 90.000,E1 243.896} C_DIS
LIN {X 0.085,Y -166.185,Z 613.345,A 0.000,B 0.000,C 90.000,E1 242.153} C_DIS
LIN {X 0.074,Y -162.955,Z 613.326,A 0.000,B 0.000,C 90.000,E1 238.663} C_DIS
LIN {X -0.102,Y -160.863,Z 613.311,A 0.000,B 0.000,C 90.000,E1 236.087} C_DIS
LIN {X 0.099,Y -157.638,Z 613.292,A 0.000,B 0.000,C 90.000,E1 232.477} C_DIS
LIN {X 0.036,Y -155.675,Z 613.277,A 0.000,B 0.000,C 90.000,E1 229.828} C_DIS
LIN {X -0.019,Y -151.942,Z 613.252,A 0.000,B 0.000,C 90.000,E1 225.364} C_DIS
LIN {X 0.102,Y -150.180,Z 613.237,A 0.000,B 0.000,C 90.000,E1 222.609} C_DIS
LIN {X 0.022,Y -146.954,Z 613.212,A 0.000,B 0.000,C 90.000,E1 218.096} C_DIS
LIN {X 0.009,Y -145.542,Z 613.196,A 0.000,B 0.000,C 90.000,E1 215.358} C_DIS
LIN {X -0.075,Y -142.938,Z 613.171,A 0.000,B 0.000,C 90.000,E1 210.797} C_DIS
LIN {X -0.017,Y -141.562,Z 613.150,A 0.000,B 0.000,C 90.000,E1 207.078} C_DIS
LIN {X 0.036,Y -139.409,Z 613.114,A 0.000,B 0.000,C 90.000,E1 200.556} C_DIS
LIN {X -0.042,Y -139.130,Z 613.104,A 0.000,B 0.000,C 90.000,E1 198.725} C_DIS
LIN {X -0.015,Y -138.350,Z 613.057,A 0.000,B 0.000,C 90.000,E1 190.310} C_DIS
LIN {X -0.028,Y -139.498,Z 613.005,A 0.000,B 0.000,C 90.000,E1 180.974} C_DIS
LIN {X 0.054,Y -141.119,Z 612.974,A 0.000,B 0.000,C 90.000,E1 175.355} C_DIS
LIN {X 0.007,Y -142.499,Z 612.959,A 0.000,B 0.000,C 90.000,E1 172.591} C_DIS
LIN {X -0.047,Y -144.753,Z 612.933,A 0.000,B 0.000,C 90.000,E1 167.993} C_DIS
LIN {X 0.045,Y -147.363,Z 612.913,A 0.000,B 0.000,C 90.000,E1 164.283} C_DIS
LIN {X -0.034,Y -150.689,Z 612.887,A 0.000,B 0.000,C 90.000,E1 159.752} C_DIS
LIN {X 0.049,Y -154.170,Z 612.867,A 0.000,B 0.000,C 90.000,E1 156.102} C_DIS
LIN {X -0.020,Y -157.604,Z 612.847,A 0.000,B 0.000,C 90.000,E1 152.538} C_DIS
LIN {X -0.070,Y -161.856,Z 612.828,A 0.000,B 0.000,C 90.000,E1 148.997} C_DIS
LIN {X -0.052,Y -166.045,Z 612.808,A 0.000,B 0.000,C 90.000,E1 145.468} C_DIS
LIN {X -0.062,Y -171.049,Z 612.789,A 0.000,B 0.000,C 90.000,E1 141.984} C_DIS
LIN {X -0.031,Y -175.921,Z 612.770,A 0.000,B 0.000,C 90.000,E1 138.528} C_DIS
LIN {X -0.039,Y -180.160,Z 612.755,A 0.000,B 0.000,C 90.000,E1 135.972} C_DIS
LIN {X -0.070,Y -185.578,Z 612.737,A 0.000,B 0.000,C 90.000,E1 132.609} C_DIS
LIN {X 0.084,Y -191.205,Z 612.719,A 0.000,B 0.000,C 90.000,E1 129.483} C_DIS
LIN {X 0.081,Y -288.400,Z 612.719,A 0.000,B 0.000,C 90.000,E1 129.483} C_DIS
LIN {X 0.036,Y -289.218,Z 612.719,A 0.000,B 0.000,C 90.000,E1 129.483} C_DIS
LIN {X -0.104,Y -294.693,Z 612.718,A 0.000,B 0.000,C 90.000,E1 129.277} C_DIS
LIN {X 0.001,Y -297.664,Z 612.717,A 0.000,B 0.000,C 90.000,E1 128.991} C_DIS
LIN {X 0.045,Y -301.375,Z 612.714,A 0.000,B 0.000,C 90.000,E1 128.463} C_DIS
LIN {X -0.010,Y -303.034,Z 612.712,A 0.000,B 0.000,C 90.000,E1 128.141} C_DIS
LIN {X -0.014,Y -304.336,Z 612.710,A 0.000,B 0.000,C 90.000,E1 127.810} C_DIS
LIN {X 0.076,Y -314.956,Z 612.690,A 0.000,B 0.000,C 90.000,E1 124.199} C_DIS
LIN {X -0.063,Y -324.890,Z 612.674,A 0.000,B 0.000,C 90.000,E1 121.337} C_DIS
LIN {X 0.027,Y -336.142,Z 612.658,A 0.000,B 0.000,C 90.000,E1 118.487} C_DIS
LIN {X -0.046,Y -348.820,Z 612.643,A 0.000,B 0.000,C 90.000,E1 115.720} C_DIS
LIN {X 0.207,Y -361.371,Z 612.629,A 0.000,B 0.000,C 90.000,E1 113.259} C_DIS
LIN {X 0.022,Y -375.227,Z 612.616,A 0.000,B 0.000,C 90.000,E1 110.918} C_DIS
LIN {X 0.047,Y -390.484,Z 612.603,A 0.000,B 0.000,C 90.000,E1 108.598} C_DIS
LIN {X 0.204,Y -407.257,Z 612.591,A 0.000,B 0.000,C 90.000,E1 106.315} C_DIS
LIN {X 0.161,Y -425.667,Z 612.579,A 0.000,B 0.000,C 90.000,E1 104.120} C_DIS
LIN {X 0.199,Y -445.520,Z 612.567,A 0.000,B 0.000,C 90.000,E1 102.007} C_DIS
LIN {X 0.168,Y -465.988,Z 612.556,A 0.000,B 0.000,C 90.000,E1 100.074} C_DIS
LIN {X 0.191,Y -471.186,Z 612.554,A 0.000,B 0.000,C 90.000,E1 99.613} C_DIS
LIN {X -0.185,Y -473.481,Z 612.552,A 0.000,B 0.000,C 90.000,E1 99.434} C_DIS
LIN {X -0.172,Y -475.215,Z 612.551,A 0.000,B 0.000,C 90.000,E1 99.208} C_DIS
LIN {X 0.160,Y -476.699,Z 612.550,A 0.000,B 0.000,C 90.000,E1 98.916} C_DIS
LIN {X 0.021,Y -477.807,Z 612.548,A 0.000,B 0.000,C 90.000,E1 98.681} C_DIS
LIN {X 0.159,Y -479.120,Z 612.545,A 0.000,B 0.000,C 90.000,E1 98.163} C_DIS
LIN {X -0.168,Y -479.416,Z 612.543,A 0.000,B 0.000,C 90.000,E1 97.701} C_DIS
LIN {X -0.011,Y -478.740,Z 612.540,A 0.000,B 0.000,C 90.000,E1 97.182} C_DIS
LIN {X 0.148,Y -476.987,Z 612.537,A 0.000,B 0.000,C 90.000,E1 96.663} C_DIS
LIN {X 0.015,Y -475.604,Z 612.536,A 0.000,B 0.000,C 90.000,E1 96.429} C_DIS
LIN {X 0.199,Y -459.526,Z 612.523,A 0.000,B 0.000,C 90.000,E1 94.131} C_DIS
LIN {X 0.211,Y -446.846,Z 612.512,A 0.000,B 0.000,C 90.000,E1 92.064} C_DIS
LIN {X -0.078,Y -435.279,Z 612.500,A 0.000,B 0.000,C 90.000,E1 90.000} C_DIS
LIN {X -0.180,Y -427.870,Z 612.493,A 0.000,B 0.000,C 90.000,E1 88.682} C_DIS
LIN {X 0.157,Y -418.510,Z 612.484,A 0.000,B 0.000,C 90.000,E1 87.020} C_DIS
LIN {X 0.162,Y -404.376,Z 612.470,A 0.000,B 0.000,C 90.000,E1 84.552} C_DIS
LIN {X -0.072,Y -390.836,Z 612.456,A 0.000,B 0.000,C 90.000,E1 82.064} C_DIS
LIN {X 0.178,Y -377.810,Z 612.442,A 0.000,B 0.000,C 90.000,E1 79.454} C_DIS
LIN {X -0.146,Y -366.631,Z 612.429,A 0.000,B 0.000,C 90.000,E1 77.173} C_DIS
LIN {X 0.061,Y -351.991,Z 612.410,A 0.000,B 0.000,C 90.000,E1 73.866} C_DIS
LIN {X -0.155,Y -337.275,Z 612.390,A 0.000,B 0.000,C 90.000,E1 70.242} C_DIS
LIN {X -0.055,Y -325.173,Z 612.371,A 0.000,B 0.000,C 90.000,E1 66.794} C_DIS
LIN {X 0.097,Y -313.276,Z 612.350,A 0.000,B 0.000,C 90.000,E1 62.948} C_DIS
LIN {X -0.103,Y -304.070,Z 612.332,A 0.000,B 0.000,C 90.000,E1 59.744} C_DIS
LIN {X 0.040,Y -295.269,Z 612.313,A 0.000,B 0.000,C 90.000,E1 56.421} C_DIS
LIN {X 0.030,Y -288.678,Z 612.299,A 0.000,B 0.000,C 90.000,E1 53.749} C_DIS
LIN {X -0.071,Y -283.807,Z 612.287,A 0.000,B 0.000,C 90.000,E1 51.743} C_DIS
LIN {X 0.085,Y -278.822,Z 612.276,A 0.000,B 0.000,C 90.000,E1 49.666} C_DIS
LIN {X -0.069,Y -273.424,Z 612.265,A 0.000,B 0.000,C 90.000,E1 47.634} C_DIS
LIN {X 0.077,Y -269.474,Z 612.257,A 0.000,B 0.000,C 90.000,E1 46.215} C_DIS
LIN {X 0.101,Y -263.061,Z 612.245,A 0.000,B 0.000,C 90.000,E1 44.109} C_DIS
LIN {X 0.038,Y -255.100,Z 612.231,A 0.000,B 0.000,C 90.000,E1 41.634} C_DIS
LIN {X 0.007,Y -245.156,Z 612.213,A 0.000,B 0.000,C 90.000,E1 38.382} C_DIS
LIN {X 0.009,Y -236.975,Z 612.197,A 0.000,B 0.000,C 90.000,E1 35.438} C_DIS
LIN {X -0.077,Y -229.635,Z 612.180,A 0.000,B 0.000,C 90.000,E1 32.467} C_DIS
LIN {X 0.113,Y -221.385,Z 612.159,A 0.000,B 0.000,C 90.000,E1 28.615} C_DIS
LIN {X 0.057,Y -215.611,Z 612.142,A 0.000,B 0.000,C 90.000,E1 25.540} C_DIS
LIN {X -0.122,Y -210.600,Z 612.125,A 0.000,B 0.000,C 90.000,E1 22.461} C_DIS
LIN {X -0.057,Y -205.457,Z 612.103,A 0.000,B 0.000,C 90.000,E1 18.489} C_DIS
LIN {X -0.017,Y -201.441,Z 612.080,A 0.000,B 0.000,C 90.000,E1 14.481} C_DIS
LIN {X 0.082,Y -197.968,Z 612.054,A 0.000,B 0.000,C 90.000,E1 9.613} C_DIS
LIN {X 0.094,Y -195.646,Z 612.013,A 0.000,B 0.000,C 90.000,E1 2.293} C_DIS
LIN {X 0.062,Y -197.442,Z 611.961,A 0.000,B 0.000,C 90.000,E1 352.996} C_DIS
LIN {X -0.086,Y -200.495,Z 611.934,A 0.000,B 0.000,C 90.000,E1 348.173} C_DIS
LIN {X 0.070,Y -204.065,Z 611.912,A 0.000,B 0.000,C 90.000,E1 344.102} C_DIS
LIN {X -0.012,Y -209.578,Z 611.885,A 0.000,B 0.000,C 90.000,E1 339.337} C_DIS
LIN {X -0.078,Y -214.977,Z 611.863,A 0.000,B 0.000,C 90.000,E1 335.409} C_DIS
LIN {X -0.090,Y -221.033,Z 611.842,A 0.000,B 0.000,C 90.000,E1 331.513} C_DIS
LIN {X -0.075,Y -227.818,Z 611.820,A 0.000,B 0.000,C 90.000,E1 327.661} C_DIS
LIN {X -0.025,Y -233.636,Z 611.803,A 0.000,B 0.000,C 90.000,E1 324.609} C_DIS
LIN {X -0.121,Y -241.322,Z 611.783,A 0.000,B 0.000,C 90.000,E1 320.884} C_DIS
LIN {X 0.081,Y -249.605,Z 611.762,A 0.000,B 0.000,C 90.000,E1 317.148} C_DIS
LIN {X -0.009,Y -258.890,Z 611.742,A 0.000,B 0.000,C 90.000,E1 313.542} C_DIS
LIN {X 0.020,Y -268.453,Z 611.724,A 0.000,B 0.000,C 90.000,E1 310.334} C_DIS
LIN {X -0.080,Y -280.669,Z 611.705,A 0.000,B 0.000,C 90.000,E1 306.870} C_DIS
LIN {X -0.005,Y -294.390,Z 611.686,A 0.000,B 0.000,C 90.000,E1 303.452} C_DIS
LIN {X 0.039,Y -309.919,Z 611.667,A 0.000,B 0.000,C 90.000,E1 300.129} C_DIS
LIN {X -0.076,Y -323.137,Z 611.653,A 0.000,B 0.000,C 90.000,E1 297.564} C_DIS
LIN {X -0.039,Y -338.766,Z 611.637,A 0.000,B 0.000,C 90.000,E1 294.719} C_DIS
LIN {X -0.089,Y -357.659,Z 611.620,A 0.000,B 0.000,C 90.000,E1 291.663} C_DIS
LIN {X 0.093,Y -376.454,Z 611.605,A 0.000,B 0.000,C 90.000,E1 288.960} C_DIS
LIN {X 0.130,Y -399.485,Z 611.589,A 0.000,B 0.000,C 90.000,E1 286.079} C_DIS
LIN {X -0.144,Y -411.071,Z 611.582,A 0.000,B 0.000,C 90.000,E1 284.717} C_DIS
LIN {X -0.106,Y -424.615,Z 611.573,A 0.000,B 0.000,C 90.000,E1 283.063} C_DIS
LIN {X 0.137,Y -433.326,Z 611.566,A 0.000,B 0.000,C 90.000,E1 281.951} C_DIS
LIN {X -0.160,Y -443.791,Z 611.559,A 0.000,B 0.000,C 90.000,E1 280.658} C_DIS
LIN {X -0.206,Y -451.758,Z 611.553,A 0.000,B 0.000,C 90.000,E1 279.613} C_DIS
LIN {X 0.111,Y -461.180,Z 611.546,A 0.000,B 0.000,C 90.000,E1 278.276} C_DIS
LIN {X 0.210,Y -468.172,Z 611.540,A 0.000,B 0.000,C 90.000,E1 277.239} C_DIS
LIN {X 0.138,Y -473.004,Z 611.536,A 0.000,B 0.000,C 90.000,E1 276.486} C_DIS
LIN {X 0.048,Y -477.154,Z 611.532,A 0.000,B 0.000,C 90.000,E1 275.739} C_DIS
LIN {X 0.186,Y -479.507,Z 611.529,A 0.000,B 0.000,C 90.000,E1 275.220} C_DIS
LIN {X -0.141,Y -481.479,Z 611.526,A 0.000,B 0.000,C 90.000,E1 274.759} C_DIS
LIN {X -0.022,Y -483.054,Z 611.524,A 0.000,B 0.000,C 90.000,E1 274.245} C_DIS
LIN {X 0.146,Y -484.348,Z 611.521,A 0.000,B 0.000,C 90.000,E1 273.726} C_DIS
LIN {X -0.191,Y -485.226,Z 611.518,A 0.000,B 0.000,C 90.000,E1 273.269} C_DIS
LIN {X -0.007,Y -485.813,Z 611.515,A 0.000,B 0.000,C 90.000,E1 272.751} C_DIS
LIN {X 0.156,Y -486.151,Z 611.513,A 0.000,B 0.000,C 90.000,E1 272.236} C_DIS
LIN {X -0.146,Y -486.166,Z 611.510,A 0.000,B 0.000,C 90.000,E1 271.776} C_DIS
LIN {X 0.025,Y -485.773,Z 611.507,A 0.000,B 0.000,C 90.000,E1 271.260} C_DIS
LIN {X 0.195,Y -484.967,Z 611.504,A 0.000,B 0.000,C 90.000,E1 270.745} C_DIS
LIN {X -0.120,Y -483.615,Z 611.502,A 0.000,B 0.000,C 90.000,E1 270.286} C_DIS
LIN {X 0.046,Y -481.711,Z 611.499,A 0.000,B 0.000,C 90.000,E1 269.771} C_DIS
LIN {X 0.201,Y -479.107,Z 611.496,A 0.000,B 0.000,C 90.000,E1 269.255} C_DIS
LIN {X -0.140,Y -475.687,Z 611.493,A 0.000,B 0.000,C 90.000,E1 268.797} C_DIS
LIN {X 0.157,Y -473.645,Z 611.492,A 0.000,B 0.000,C 90.000,E1 268.511} C_DIS
LIN {X -0.194,Y -468.630,Z 611.489,A 0.000,B 0.000,C 90.000,E1 268.051} C_DIS
LIN {X 0.088,Y -465.672,Z 611.488,A 0.000,B 0.000,C 90.000,E1 267.764} C_DIS
LIN {X 0.130,Y -462.581,Z 611.486,A 0.000,B 0.000,C 90.000,E1 267.535} C_DIS
LIN {X 0.170,Y -459.085,Z 611.485,A 0.000,B 0.000,C 90.000,E1 267.306} C_DIS
LIN {X 0.002,Y -452.019,Z 611.483,A 0.000,B 0.000,C 90.000,E1 266.963} C_DIS
LIN {X 0.011,Y -444.747,Z 611.482,A 0.000,B 0.000,C 90.000,E1 266.674} C_DIS
LIN {X -0.020,Y -436.864,Z 611.480,A 0.000,B 0.000,C 90.000,E1 266.445} C_DIS
LIN {X -0.043,Y -428.134,Z 611.479,A 0.000,B 0.000,C 90.000,E1 266.274} C_DIS
LIN {X -0.071,Y -418.464,Z 611.479,A 0.000,B 0.000,C 90.000,E1 266.159} C_DIS
LIN {X -0.022,Y -407.451,Z 611.478,A 0.000,B 0.000,C 90.000,E1 266.102} C_DIS
LIN {X -0.042,Y -180.924,Z 611.478,A 0.000,B 0.000,C 90.000,E1 266.102} C_DIS
LIN {X -0.048,Y -180.899,Z 611.473,A 0.000,B 0.000,C 90.000,E1 265.241} C_DIS
LIN {X 0.080,Y -180.210,Z 611.464,A 0.000,B 0.000,C 90.000,E1 263.514} C_DIS
LIN {X 0.031,Y -179.031,Z 611.445,A 0.000,B 0.000,C 90.000,E1 260.151} C_DIS
LIN {X -0.082,Y -178.685,Z 611.441,A 0.000,B 0.000,C 90.000,E1 259.342} C_DIS
LIN {X 0.029,Y -175.735,Z 611.412,A 0.000,B 0.000,C 90.000,E1 254.212} C_DIS
LIN {X 0.024,Y -171.918,Z 611.384,A 0.000,B 0.000,C 90.000,E1 249.082} C_DIS
LIN {X 0.000,Y -171.289,Z 611.379,A 0.000,B 0.000,C 90.000,E1 248.230} C_DIS
LIN {X 0.045,Y -167.553,Z 611.355,A 0.000,B 0.000,C 90.000,E1 243.896} C_DIS
LIN {X 0.058,Y -166.176,Z 611.345,A 0.000,B 0.000,C 90.000,E1 242.153} C_DIS
LIN {X 0.048,Y -162.948,Z 611.326,A 0.000,B 0.000,C 90.000,E1 238.663} C_DIS
LIN {X 0.096,Y -160.854,Z 611.311,A 0.000,B 0.000,C 90.000,E1 236.008} C_DIS
LIN {X 0.073,Y -157.630,Z 611.292,A 0.000,B 0.000,C 90.000,E1 232.477} C_DIS
LIN {X 0.011,Y -155.667,Z 611.277,A 0.000,B 0.000,C 90.000,E1 229.828} C_DIS
LIN {X 0.063,Y -151.935,Z 611.252,A 0.000,B 0.000,C 90.000,E1 225.324} C_DIS
LIN {X 0.078,Y -150.173,Z 611.237,A 0.000,B 0.000,C 90.000,E1 222.609} C_DIS
LIN {X -0.002,Y -146.949,Z 611.212,A 0.000,B 0.000,C 90.000,E1 218.096} C_DIS
LIN {X -0.014,Y -145.537,Z 611.196,A 0.000,B 0.000,C 90.000,E1 215.358} C_DIS
LIN {X 0.024,Y -142.933,Z 611.171,A 0.000,B 0.000,C 90.000,E1 210.747} C_DIS
LIN {X 0.024,Y -141.556,Z 611.150,A 0.000,B 0.000,C 90.000,E1 207.052} C_DIS
LIN {X 0.013,Y -139.408,Z 611.114,A 0.000,B 0.000,C 90.000,E1 200.556} C_DIS
LIN {X -0.066,Y -139.128,Z 611.104,A 0.000,B 0.000,C 90.000,E1 198.725} C_DIS
LIN {X -0.039,Y -138.351,Z 611.057,A 0.000,B 0.000,C 90.000,E1 190.310} C_DIS
LIN {X -0.051,Y -139.499,Z 611.005,A 0.000,B 0.000,C 90.000,E1 180.974} C_DIS
LIN {X 0.029,Y -141.123,Z 610.974,A 0.000,B 0.000,C 90.000,E1 175.355} C_DIS
LIN {X -0.018,Y -142.503,Z 610.959,A 0.000,B 0.000,C 90.000,E1 172.591} C_DIS
LIN {X 0.071,Y -144.760,Z 610.933,A 0.000,B 0.000,C 90.000,E1 167.937} C_DIS
LIN {X 0.020,Y -147.370,Z 610.913,A 0.000,B 0.000,C 90.000,E1 164.283} C_DIS
LIN {X -0.059,Y -150.697,Z 610.887,A 0.000,B 0.000,C 90.000,E1 159.752} C_DIS
LIN {X 0.025,Y -154.179,Z 610.867,A 0.000,B 0.000,C 90.000,E1 156.102} C_DIS
LIN {X -0.045,Y -157.614,Z 610.847,A 0.000,B 0.000,C 90.000,E1 152.538} C_DIS
LIN {X 0.043,Y -161.867,Z 610.828,A 0.000,B 0.000,C 90.000,E1 148.948} C_DIS
LIN {X -0.079,Y -166.058,Z 610.808,A 0.000,B 0.000,C 90.000,E1 145.468} C_DIS
LIN {X -0.088,Y -171.063,Z 610.789,A 0.000,B 0.000,C 90.000,E1 141.984} C_DIS
LIN {X -0.059,Y -175.935,Z 610.769,A 0.000,B 0.000,C 90.000,E1 138.528} C_DIS
LIN {X -0.067,Y -180.176,Z 610.755,A 0.000,B 0.000,C 90.000,E1 135.972} C_DIS
LIN {X -0.099,Y -185.592,Z 610.737,A 0.000,B 0.000,C 90.000,E1 132.609} C_DIS
LIN {X 0.054,Y -191.219,Z 610.719,A 0.000,B 0.000,C 90.000,E1 129.483} C_DIS
LIN {X 0.037,Y -288.203,Z 610.719,A 0.000,B 0.000,C 90.000,E1 129.483} C_DIS
LIN {X -0.008,Y -289.140,Z 610.719,A 0.000,B 0.000,C 90.000,E1 129.483} C_DIS
LIN {X -0.148,Y -294.680,Z 610.718,A 0.000,B 0.000,C 90.000,E1 129.277} C_DIS
LIN {X -0.028,Y -297.629,Z 610.717,A 0.000,B 0.000,C 90.000,E1 128.991} C_DIS
LIN {X 0.026,Y -301.346,Z 610.714,A 0.000,B 0.000,C 90.000,E1 128.463} C_DIS
LIN {X -0.029,Y -303.013,Z 610.712,A 0.000,B 0.000,C 90.000,E1 128.141} C_DIS
LIN {X -0.034,Y -304.321,Z 610.710,A 0.000,B 0.000,C 90.000,E1 127.810} C_DIS
LIN {X 0.054,Y -314.947,Z 610.690,A 0.000,B 0.000,C 90.000,E1 124.199} C_DIS
LIN {X -0.084,Y -324.883,Z 610.674,A 0.000,B 0.000,C 90.000,E1 121.337} C_DIS
LIN {X 0.004,Y -336.137,Z 610.658,A 0.000,B 0.000,C 90.000,E1 118.487} C_DIS
LIN {X -0.070,Y -348.815,Z 610.643,A 0.000,B 0.000,C 90.000,E1 115.720} C_DIS
LIN {X 0.183,Y -361.369,Z 610.629,A 0.000,B 0.000,C 90.000,E1 113.259} C_DIS
LIN {X -0.003,Y -375.227,Z 610.616,A 0.000,B 0.000,C 90.000,E1 110.918} C_DIS
LIN {X 0.020,Y -390.487,Z 610.603,A 0.000,B 0.000,C 90.000,E1 108.598} C_DIS
LIN {X 0.176,Y -407.261,Z 610.591,A 0.000,B 0.000,C 90.000,E1 106.315} C_DIS
LIN {X 0.131,Y -425.674,Z 610.579,A 0.000,B 0.000,C 90.000,E1 104.120} C_DIS
LIN {X 0.169,Y -445.528,Z 610.567,A 0.000,B 0.000,C 90.000,E1 102.007} C_DIS
LIN {X 0.139,Y -465.997,Z 610.556,A 0.000,B 0.000,C 90.000,E1 100.074} C_DIS
LIN {X 0.162,Y -471.197,Z 610.554,A 0.000,B 0.000,C 90.000,E1 99.613} C_DIS
LIN {X 0.253,Y -473.509,Z 610.552,A 0.000,B 0.000,C 90.000,E1 99.378} C_DIS
LIN {X -0.202,Y -475.259,Z 610.551,A 0.000,B 0.000,C 90.000,E1 99.208} C_DIS
LIN {X 0.131,Y -476.755,Z 610.550,A 0.000,B 0.000,C 90.000,E1 98.916} C_DIS
LIN {X -0.009,Y -477.873,Z 610.548,A 0.000,B 0.000,C 90.000,E1 98.681} C_DIS
LIN {X 0.131,Y -479.202,Z 610.545,A 0.000,B 0.000,C 90.000,E1 98.163} C_DIS
LIN {X -0.196,Y -479.510,Z 610.543,A 0.000,B 0.000,C 90.000,E1 97.701} C_DIS
LIN {X -0.039,Y -478.848,Z 610.540,A 0.000,B 0.000,C 90.000,E1 97.182} C_DIS
LIN {X 0.120,Y -477.110,Z 610.537,A 0.000,B 0.000,C 90.000,E1 96.663} C_DIS
LIN {X -0.011,Y -475.739,Z 610.536,A 0.000,B 0.000,C 90.000,E1 96.429} C_DIS
LIN {X 0.177,Y -459.646,Z 610.523,A 0.000,B 0.000,C 90.000,E1 94.131} C_DIS
LIN {X -0.016,Y -448.434,Z 610.513,A 0.000,B 0.000,C 90.000,E1 92.350} C_DIS
LIN {X -0.095,Y -435.369,Z 610.500,A 0.000,B 0.000,C 90.000,E1 90.000} C_DIS
LIN {X -0.195,Y -427.945,Z 610.493,A 0.000,B 0.000,C 90.000,E1 88.682} C_DIS
LIN {X 0.143,Y -418.582,Z 610.484,A 0.000,B 0.000,C 90.000,E1 87.020} C_DIS
LIN {X 0.151,Y -404.444,Z 610.470,A 0.000,B 0.000,C 90.000,E1 84.552} C_DIS
LIN {X -0.082,Y -390.906,Z 610.456,A 0.000,B 0.000,C 90.000,E1 82.064} C_DIS
LIN {X 0.171,Y -377.872,Z 610.442,A 0.000,B 0.000,C 90.000,E1 79.454} C_DIS
LIN {X -0.152,Y -366.677,Z 610.429,A 0.000,B 0.000,C 90.000,E1 77.173} C_DIS
LIN {X 0.077,Y -354.577,Z 610.414,A 0.000,B 0.000,C 90.000,E1 74.464} C_DIS
LIN {X -0.076,Y -343.256,Z 610.399,A 0.000,B 0.000,C 90.000,E1 71.764} C_DIS
LIN {X 0.064,Y -329.501,Z 610.378,A 0.000,B 0.000,C 90.000,E1 68.028} C_DIS
LIN {X -0.179,Y -317.185,Z 610.357,A 0.000,B 0.000,C 90.000,E1 64.280} C_DIS
LIN {X -0.123,Y -307.815,Z 610.339,A 0.000,B 0.000,C 90.000,E1 61.051} C_DIS
LIN {X 0.080,Y -298.820,Z 610.321,A 0.000,B 0.000,C 90.000,E1 57.740} C_DIS
LIN {X 0.134,Y -290.380,Z 610.302,A 0.000,B 0.000,C 90.000,E1 54.402} C_DIS
LIN {X -0.059,Y -283.878,Z 610.287,A 0.000,B 0.000,C 90.000,E1 51.743} C_DIS
LIN {X -0.082,Y -278.897,Z 610.276,A 0.000,B 0.000,C 90.000,E1 49.703} C_DIS
LIN {X -0.054,Y -273.498,Z 610.265,A 0.000,B 0.000,C 90.000,E1 47.634} C_DIS
LIN {X 0.091,Y -269.543,Z 610.257,A 0.000,B 0.000,C 90.000,E1 46.215} C_DIS
LIN {X -0.130,Y -264.207,Z 610.247,A 0.000,B 0.000,C 90.000,E1 44.514} C_DIS
LIN {X -0.030,Y -257.446,Z 610.235,A 0.000,B 0.000,C 90.000,E1 42.366} C_DIS
LIN {X 0.001,Y -247.364,Z 610.217,A 0.000,B 0.000,C 90.000,E1 39.116} C_DIS
LIN {X 0.054,Y -238.978,Z 610.201,A 0.000,B 0.000,C 90.000,E1 36.171} C_DIS
LIN {X -0.042,Y -231.445,Z 610.184,A 0.000,B 0.000,C 90.000,E1 33.214} C_DIS
LIN {X -0.118,Y -224.594,Z 610.168,A 0.000,B 0.000,C 90.000,E1 30.207} C_DIS
LIN {X -0.080,Y -218.427,Z 610.151,A 0.000,B 0.000,C 90.000,E1 27.129} C_DIS
LIN {X -0.015,Y -213.034,Z 610.133,A 0.000,B 0.000,C 90.000,E1 24.003} C_DIS
LIN {X -0.034,Y -208.430,Z 610.116,A 0.000,B 0.000,C 90.000,E1 20.865} C_DIS
LIN {X 0.087,Y -203.717,Z 610.094,A 0.000,B 0.000,C 90.000,E1 16.858} C_DIS
LIN {X 0.010,Y -199.559,Z 610.067,A 0.000,B 0.000,C 90.000,E1 12.063} C_DIS
LIN {X 0.080,Y -196.527,Z 610.036,A 0.000,B 0.000,C 90.000,E1 6.372} C_DIS
LIN {X 0.063,Y -197.467,Z 609.961,A 0.000,B 0.000,C 90.000,E1 352.996} C_DIS
LIN {X -0.084,Y -200.557,Z 609.934,A 0.000,B 0.000,C 90.000,E1 348.173} C_DIS
LIN {X -0.006,Y -204.958,Z 609.907,A 0.000,B 0.000,C 90.000,E1 343.323} C_DIS
LIN {X -0.006,Y -209.621,Z 609.885,A 0.000,B 0.000,C 90.000,E1 339.337} C_DIS
LIN {X -0.071,Y -215.006,Z 609.863,A 0.000,B 0.000,C 90.000,E1 335.409} C_DIS
LIN {X -0.083,Y -221.066,Z 609.842,A 0.000,B 0.000,C 90.000,E1 331.513} C_DIS
LIN {X -0.066,Y -227.846,Z 609.820,A 0.000,B 0.000,C 90.000,E1 327.661} C_DIS
LIN {X -0.014,Y -233.653,Z 609.803,A 0.000,B 0.000,C 90.000,E1 324.609} C_DIS
LIN {X -0.110,Y -241.308,Z 609.783,A 0.000,B 0.000,C 90.000,E1 320.884} C_DIS
LIN {X 0.091,Y -249.563,Z 609.762,A 0.000,B 0.000,C 90.000,E1 317.148} C_DIS
LIN {X 0.001,Y -258.840,Z 609.742,A 0.000,B 0.000,C 90.000,E1 313.542} C_DIS
LIN {X 0.028,Y -268.396,Z 609.724,A 0.000,B 0.000,C 90.000,E1 310.334} C_DIS
LIN {X -0.073,Y -280.598,Z 609.705,A 0.000,B 0.000,C 90.000,E1 306.870} C_DIS
LIN {X 0.012,Y -292.842,Z 609.688,A 0.000,B 0.000,C 90.000,E1 303.785} C_DIS
LIN {X 0.003,Y -308.234,Z 609.669,A 0.000,B 0.000,C 90.000,E1 300.463} C_DIS
LIN {X 0.131,Y -321.356,Z 609.655,A 0.000,B 0.000,C 90.000,E1 297.847} C_DIS
LIN {X -0.019,Y -336.845,Z 609.639,A 0.000,B 0.000,C 90.000,E1 295.027} C_DIS
LIN {X -0.036,Y -353.652,Z 609.624,A 0.000,B 0.000,C 90.000,E1 292.259} C_DIS
LIN {X -0.105,Y -372.089,Z 609.609,A 0.000,B 0.000,C 90.000,E1 289.577} C_DIS
LIN {X 0.069,Y -387.729,Z 609.597,A 0.000,B 0.000,C 90.000,E1 287.511} C_DIS
LIN {X -0.206,Y -401.802,Z 609.588,A 0.000,B 0.000,C 90.000,E1 285.843} C_DIS
LIN {X 0.056,Y -413.305,Z 609.580,A 0.000,B 0.000,C 90.000,E1 284.411} C_DIS
LIN {X 0.039,Y -426.867,Z 609.571,A 0.000,B 0.000,C 90.000,E1 282.771} C_DIS
LIN {X 0.074,Y -437.606,Z 609.564,A 0.000,B 0.000,C 90.000,E1 281.422} C_DIS
LIN {X -0.246,Y -447.897,Z 609.556,A 0.000,B 0.000,C 90.000,E1 280.141} C_DIS
LIN {X -0.168,Y -455.602,Z 609.550,A 0.000,B 0.000,C 90.000,E1 279.086} C_DIS
LIN {X -0.143,Y -462.927,Z 609.545,A 0.000,B 0.000,C 90.000,E1 278.049} C_DIS
LIN {X 0.036,Y -469.786,Z 609.539,A 0.000,B 0.000,C 90.000,E1 277.004} C_DIS
LIN {X -0.084,Y -474.356,Z 609.535,A 0.000,B 0.000,C 90.000,E1 276.258} C_DIS
LIN {X -0.156,Y -478.253,Z 609.531,A 0.000,B 0.000,C 90.000,E1 275.511} C_DIS
LIN {X 0.173,Y -479.434,Z 609.529,A 0.000,B 0.000,C 90.000,E1 275.220} C_DIS
LIN {X -0.155,Y -481.430,Z 609.526,A 0.000,B 0.000,C 90.000,E1 274.759} C_DIS
LIN {X -0.037,Y -483.059,Z 609.524,A 0.000,B 0.000,C 90.000,E1 274.245} C_DIS
LIN {X 0.132,Y -484.306,Z 609.521,A 0.000,B 0.000,C 90.000,E1 273.726} C_DIS
LIN {X -0.205,Y -485.183,Z 609.518,A 0.000,B 0.000,C 90.000,E1 273.269} C_DIS
LIN {X -0.023,Y -485.803,Z 609.515,A 0.000,B 0.000,C 90.000,E1 272.751} C_DIS
LIN {X 0.140,Y -486.134,Z 609.513,A 0.000,B 0.000,C 90.000,E1 272.236} C_DIS
LIN {X -0.161,Y -486.195,Z 609.510,A 0.000,B 0.000,C 90.000,E1 271.776} C_DIS
LIN {X 0.008,Y -485.823,Z 609.507,A 0.000,B 0.000,C 90.000,E1 271.260} C_DIS
LIN {X 0.181,Y -484.989,Z 609.504,A 0.000,B 0.000,C 90.000,E1 270.745} C_DIS
LIN {X -0.134,Y -483.669,Z 609.502,A 0.000,B 0.000,C 90.000,E1 270.286} C_DIS
LIN {X 0.031,Y -481.731,Z 609.499,A 0.000,B 0.000,C 90.000,E1 269.771} C_DIS
LIN {X -0.132,Y -480.566,Z 609.497,A 0.000,B 0.000,C 90.000,E1 269.542} C_DIS
LIN {X 0.016,Y -477.510,Z 609.495,A 0.000,B 0.000,C 90.000,E1 269.026} C_DIS
LIN {X 0.142,Y -473.676,Z 609.492,A 0.000,B 0.000,C 90.000,E1 268.511} C_DIS
LIN {X -0.036,Y -471.317,Z 609.490,A 0.000,B 0.000,C 90.000,E1 268.282} C_DIS
LIN {X 0.075,Y -465.651,Z 609.488,A 0.000,B 0.000,C 90.000,E1 267.764} C_DIS
LIN {X 0.127,Y -462.587,Z 609.486,A 0.000,B 0.000,C 90.000,E1 267.535} C_DIS
LIN {X 0.178,Y -459.084,Z 609.485,A 0.000,B 0.000,C 90.000,E1 267.306} C_DIS
LIN {X 0.030,Y -452.102,Z 609.483,A 0.000,B 0.000,C 90.000,E1 266.963} C_DIS
LIN {X 0.008,Y -444.717,Z 609.482,A 0.000,B 0.000,C 90.000,E1 266.674} C_DIS
LIN {X 0.000,Y -436.933,Z 609.480,A 0.000,B 0.000,C 90.000,E1 266.445} C_DIS
LIN {X -0.028,Y -428.135,Z 609.479,A 0.000,B 0.000,C 90.000,E1 266.274} C_DIS
LIN {X -0.044,Y -418.557,Z 609.479,A 0.000,B 0.000,C 90.000,E1 266.159} C_DIS
LIN {X 0.008,Y -410.107,Z 609.478,A 0.000,B 0.000,C 90.000,E1 266.102} C_DIS
LIN {X -0.028,Y -180.924,Z 609.478,A 0.000,B 0.000,C 90.000,E1 266.102} C_DIS
LIN {X -0.034,Y -180.898,Z 609.474,A 0.000,B 0.000,C 90.000,E1 265.241} C_DIS
LIN {X -0.085,Y -180.213,Z 609.464,A 0.000,B 0.000,C 90.000,E1 263.571} C_DIS
LIN {X 0.045,Y -179.033,Z 609.445,A 0.000,B 0.000,C 90.000,E1 260.151} C_DIS
LIN {X -0.068,Y -178.688,Z 609.441,A 0.000,B 0.000,C 90.000,E1 259.342} C_DIS
LIN {X 0.043,Y -175.738,Z 609.412,A 0.000,B 0.000,C 90.000,E1 254.212} C_DIS
LIN {X 0.038,Y -171.921,Z 609.384,A 0.000,B 0.000,C 90.000,E1 249.082} C_DIS
LIN {X 0.013,Y -171.293,Z 609.379,A 0.000,B 0.000,C 90.000,E1 248.230} C_DIS
LIN {X 0.059,Y -167.557,Z 609.355,A 0.000,B 0.000,C 90.000,E1 243.896} C_DIS
LIN {X 0.072,Y -166.181,Z 609.345,A 0.000,B 0.000,C 90.000,E1 242.153} C_DIS
LIN {X 0.062,Y -162.951,Z 609.326,A 0.000,B 0.000,C 90.000,E1 238.663} C_DIS
LIN {X 0.109,Y -160.858,Z 609.311,A 0.000,B 0.000,C 90.000,E1 236.008} C_DIS
LIN {X 0.086,Y -157.634,Z 609.292,A 0.000,B 0.000,C 90.000,E1 232.477} C_DIS
LIN {X 0.024,Y -155.672,Z 609.277,A 0.000,B 0.000,C 90.000,E1 229.828} C_DIS
LIN {X 0.075,Y -151.939,Z 609.252,A 0.000,B 0.000,C 90.000,E1 225.324} C_DIS
LIN {X 0.091,Y -150.176,Z 609.237,A 0.000,B 0.000,C 90.000,E1 222.609} C_DIS
LIN {X 0.011,Y -146.952,Z 609.212,A 0.000,B 0.000,C 90.000,E1 218.096} C_DIS
LIN {X -0.002,Y -145.539,Z 609.196,A 0.000,B 0.000,C 90.000,E1 215.358} C_DIS
LIN {X 0.037,Y -142.935,Z 609.171,A 0.000,B 0.000,C 90.000,E1 210.747} C_DIS
LIN {X -0.029,Y -141.559,Z 609.150,A 0.000,B 0.000,C 90.000,E1 207.078} C_DIS
LIN {X 0.024,Y -139.409,Z 609.114,A 0.000,B 0.000,C 90.000,E1 200.556} C_DIS
LIN {X -0.054,Y -139.129,Z 609.104,A 0.000,B 0.000,C 90.000,E1 198.725} C_DIS
LIN {X -0.026,Y -138.350,Z 609.057,A 0.000,B 0.000,C 90.000,E1 190.310} C_DIS
LIN {X -0.039,Y -139.498,Z 609.005,A 0.000,B 0.000,C 90.000,E1 180.974} C_DIS
LIN {X 0.042,Y -141.121,Z 608.974,A 0.000,B 0.000,C 90.000,E1 175.355} C_DIS
LIN {X -0.005,Y -142.500,Z 608.959,A 0.000,B 0.000,C 90.000,E1 172.591} C_DIS
LIN {X -0.058,Y -144.756,Z 608.933,A 0.000,B 0.000,C 90.000,E1 167.993} C_DIS
LIN {X 0.032,Y -147.366,Z 608.913,A 0.000,B 0.000,C 90.000,E1 164.283} C_DIS
LIN {X -0.045,Y -150.694,Z 608.887,A 0.000,B 0.000,C 90.000,E1 159.752} C_DIS
LIN {X 0.038,Y -154.174,Z 608.867,A 0.000,B 0.000,C 90.000,E1 156.102} C_DIS
LIN {X -0.033,Y -157.608,Z 608.847,A 0.000,B 0.000,C 90.000,E1 152.538} C_DIS
LIN {X 0.056,Y -161.861,Z 608.828,A 0.000,B 0.000,C 90.000,E1 148.948} C_DIS
LIN {X -0.065,Y -166.052,Z 608.808,A 0.000,B 0.000,C 90.000,E1 145.468} C_DIS
LIN {X -0.075,Y -171.056,Z 608.789,A 0.000,B 0.000,C 90.000,E1 141.984} C_DIS
LIN {X -0.045,Y -175.928,Z 608.770,A 0.000,B 0.000,C 90.000,E1 138.528} C_DIS
LIN {X -0.052,Y -180.168,Z 608.755,A 0.000,B 0.000,C 90.000,E1 135.972} C_DIS
LIN {X -0.084,Y -185.584,Z 608.737,A 0.000,B 0.000,C 90.000,E1 132.609} C_DIS
LIN {X 0.007,Y -191.242,Z 608.719,A 0.000,B 0.000,C 90.000,E1 129.483} C_DIS
LIN {X -0.029,Y -288.564,Z 608.719,A 0.000,B 0.000,C 90.000,E1 129.483} C_DIS
LIN {X 0.076,Y -290.053,Z 608.719,A 0.000,B 0.000,C 90.000,E1 129.439} C_DIS
LIN {X -0.125,Y -294.473,Z 608.718,A 0.000,B 0.000,C 90.000,E1 129.277} C_DIS
LIN {X -0.110,Y -297.684,Z 608.716,A 0.000,B 0.000,C 90.000,E1 128.991} C_DIS
LIN {X -0.032,Y -301.356,Z 608.714,A 0.000,B 0.000,C 90.000,E1 128.463} C_DIS
LIN {X 0.151,Y -303.023,Z 608.712,A 0.000,B 0.000,C 90.000,E1 128.096} C_DIS
LIN {X -0.092,Y -304.330,Z 608.710,A 0.000,B 0.000,C 90.000,E1 127.810} C_DIS
LIN {X -0.006,Y -314.962,Z 608.690,A 0.000,B 0.000,C 90.000,E1 124.199} C_DIS
LIN {X -0.146,Y -324.901,Z 608.674,A 0.000,B 0.000,C 90.000,E1 121.337} C_DIS
LIN {X -0.059,Y -336.160,Z 608.658,A 0.000,B 0.000,C 90.000,E1 118.487} C_DIS
LIN {X -0.135,Y -348.844,Z 608.643,A 0.000,B 0.000,C 90.000,E1 115.720} C_DIS
LIN {X 0.117,Y -361.403,Z 608.629,A 0.000,B 0.000,C 90.000,E1 113.259} C_DIS
LIN {X -0.071,Y -375.266,Z 608.616,A 0.000,B 0.000,C 90.000,E1 110.918} C_DIS
LIN {X -0.049,Y -390.532,Z 608.603,A 0.000,B 0.000,C 90.000,E1 108.598} C_DIS
LIN {X 0.105,Y -407.314,Z 608.591,A 0.000,B 0.000,C 90.000,E1 106.315} C_DIS
LIN {X 0.058,Y -425.733,Z 608.578,A 0.000,B 0.000,C 90.000,E1 104.120} C_DIS
LIN {X 0.097,Y -445.591,Z 608.567,A 0.000,B 0.000,C 90.000,E1 102.007} C_DIS
LIN {X 0.069,Y -466.064,Z 608.556,A 0.000,B 0.000,C 90.000,E1 100.074} C_DIS
LIN {X 0.093,Y -471.263,Z 608.553,A 0.000,B 0.000,C 90.000,E1 99.613} C_DIS
LIN {X 0.184,Y -473.582,Z 608.552,A 0.000,B 0.000,C 90.000,E1 99.378} C_DIS
LIN {X 0.198,Y -475.336,Z 608.551,A 0.000,B 0.000,C 90.000,E1 99.151} C_DIS
LIN {X 0.061,Y -476.836,Z 608.550,A 0.000,B 0.000,C 90.000,E1 98.916} C_DIS
LIN {X -0.078,Y -477.957,Z 608.548,A 0.000,B 0.000,C 90.000,E1 98.681} C_DIS
LIN {X 0.062,Y -479.292,Z 608.545,A 0.000,B 0.000,C 90.000,E1 98.163} C_DIS
LIN {X 0.211,Y -479.607,Z 608.543,A 0.000,B 0.000,C 90.000,E1 97.644} C_DIS
LIN {X -0.107,Y -478.951,Z 608.540,A 0.000,B 0.000,C 90.000,E1 97.182} C_DIS
LIN {X 0.054,Y -477.220,Z 608.537,A 0.000,B 0.000,C 90.000,E1 96.663} C_DIS
LIN {X -0.079,Y -475.853,Z 608.536,A 0.000,B 0.000,C 90.000,E1 96.429} C_DIS
LIN {X 0.115,Y -459.719,Z 608.523,A 0.000,B 0.000,C 90.000,E1 94.131} C_DIS
LIN {X 0.133,Y -446.985,Z 608.512,A 0.000,B 0.000,C 90.000,E1 92.064} C_DIS
LIN {X 0.011,Y -433.980,Z 608.498,A 0.000,B 0.000,C 90.000,E1 89.714} C_DIS
LIN {X -0.108,Y -426.458,Z 608.491,A 0.000,B 0.000,C 90.000,E1 88.396} C_DIS
LIN {X -0.195,Y -417.030,Z 608.482,A 0.000,B 0.000,C 90.000,E1 86.788} C_DIS
LIN {X 0.193,Y -402.942,Z 608.468,A 0.000,B 0.000,C 90.000,E1 84.261} C_DIS
LIN {X -0.070,Y -388.008,Z 608.453,A 0.000,B 0.000,C 90.000,E1 81.489} C_DIS
LIN {X 0.145,Y -376.474,Z 608.440,A 0.000,B 0.000,C 90.000,E1 79.162} C_DIS
LIN {X 0.146,Y -365.308,Z 608.427,A 0.000,B 0.000,C 90.000,E1 76.825} C_DIS
LIN {X 0.080,Y -353.291,Z 608.412,A 0.000,B 0.000,C 90.000,E1 74.157} C_DIS
LIN {X -0.093,Y -340.851,Z 608.395,A 0.000,B 0.000,C 90.000,E1 71.148} C_DIS
LIN {X -0.029,Y -327.403,Z 608.374,A 0.000,B 0.000,C 90.000,E1 67.411} C_DIS
LIN {X 0.072,Y -317.262,Z 608.357,A 0.000,B 0.000,C 90.000,E1 64.229} C_DIS
